	3:
		bTimer1															:= TRUE;
		bPass1															:= steam_bypass_valve_clear;
		bPass2															:= steam_iso_valve_clear;
		bPass3															:= product_iso_valve_clear;
		bPass4															:= r1.fan_vfd_output = 0;
		bPass5															:= P_U01.vacuum_pres_control_valve_closed;
		bPass6															:= P_U01.steam_flow_control_valve_closed;
		bPass7															:= P_U01.product_line_ambient_valve_clear;
		bPass8															:= P_U01.vacuum_pump_bypass_valve_clear;
		bPass9															:= P_U01.vacuum_pump_inlet_valve_clear;
		IF bPass1 AND bPass2 AND bPass3 AND bPass4 AND bPass5 AND bPass6 AND bPass7 AND bPass8 AND bPass9 THEN
			bTimer1														:= FALSE;
			rTime1														:= _SECONDS * 60;
			i6Step														:= i6Step + 1;
		ELSIF tonTimer1.Q THEN
			bTimer1														:= FALSE;
			sReactorError												:= SEL(bPass1,'Steam Bypass Valve Error RS XV08', '');
			sReactorError												:= SEL(bPass2, gsSteamIsoValveError, sReactorError);
			sReactorError												:= SEL(bPass3, gsProductIsoValveError, sReactorError);
			sReactorError												:= SEL(bPass4, 'Fan VFD SP Error', sReactorError);
			sUtilityError												:= SEL(bPass5, gsVacuumPressureControlValveError, '');
			sUtilityError												:= SEL(bPass6, gsSteamFlowConrolValveError, sUtilityError);
			sUtilityError												:= SEL(bPass7, gsProductLineAmbientValveError, sUtilityError);
			sUtilityError												:= SEL(bPass8, gsVacuumPumpBypassValveError, sUtilityError);
			sUtilityError												:= SEL(bPass9, gsVacuumPumpInletValveError, sUtilityError);
		END_IF
		
	4:
		bTimer1															:= TRUE;
		bPass1															:= r1.reactor_pres > P_M01.SP_evacuation_ideal_pressure;
		bPass2															:= NOT reactor_drain_vessel_lsh;
		bPass3															:= NOT P_U01.product_condensate_drum_lsh;
//		bPass4															:= P_U01.vacuum_separator_level > P_U01.SP_vacuum_separator_level_low;
		IF bPass1 AND bPass2 AND bPass3  THEN
			bTimer1														:= FALSE;
			cycle_stage													:= 'evacuation.starting';
			P_U01.drainage_on											:= FALSE;											
			i6Step														:= i6Step + 1;
		ELSIF tonTimer1.Q THEN
			bTimer1														:= FALSE;
			sReactorError												:= SEL(bPass1, gsReactorPressureTooLowError, '');
			sReactorError												:= SEL(bPass2, gsReactorDrainError, sReactorError);
			sUtilityError												:= SEL(bPass3, gsProductCondensateDrumLshError, '');
		END_IF
	
	5:
		
			rTime1														:= _CLAMP_ACTUATION_TIMEOUT;
			P_U01.vacuum_liquid_pump									:= TRUE;											
			P_U01.vacuum_liquid_loop_fan								:= TRUE;
			retract_clamps												:= TRUE;											
			i6Step														:= i6Step + 1;
		
	6:
		bTimer1															:= TRUE;
		IF inlet_clamps_retracted AND outlet_clamps_retracted THEN
			bTimer1														:= FALSE;
			close_doors													:= TRUE;											
			rTime1														:= _DOOR_ACTUATION_TIMEOUT;
			i6Step														:= i6Step + 1;
		ELSIF tonTimer1.Q THEN
			bTimer1														:= FALSE;
			sReactorError												:= SEL(inlet_clamps_retracted, gsInletDoorClampsRetractedError, '');
			sReactorError												:= SEL(outlet_clamps_retracted, gsOutletDoorClampsRetractedError, sReactorError);
		END_IF

	7:
		bTimer1															:= TRUE;
		IF inlet_doors_closed AND outlet_doors_closed THEN
			bTimer1														:= FALSE;
			extend_clamps												:= TRUE;											
			rTime1														:= 30 * _SECONDS;
			i6Step														:= i6Step + 1;
		ELSIF tonTimer1.Q THEN
			sReactorError												:= gsDoorsNotClosedError;
			bTimer1														:= FALSE;
		END_IF

	8:
		cycle_stage														:= 'evacuation.vacuum_init';
		bTimer1															:= TRUE;
		bPass1															:= P_U01.vacuum_pump_water_flow > P_U01.SP_minimum_vacuum_cooling_loop_flow;
		bPass2															:= P_U01.vacuum_pump_water_temp_1 < P_U01.SP_max_vacuum_cooling_loop_temp;
		IF bPass1 AND bPass2 THEN																							
			bTimer1														:= FALSE;
			cycle_stage													:= 'evacuation.evacuation';
			P_U01.dead_air_inlet_valve									:= TRUE;
			P_U01.vacuum_pump											:= TRUE;
			rTime1														:= 20 * _SECONDS;
			i6Step														:= i6Step + 1;
		ELSIF tonTimer1.Q THEN
			bTimer1														:= FALSE;
			sUtilityError												:= SEL(bPass1, gsVacuumCoolingLoopFlowError, '');
			sUtilityError												:= SEL(bPass2, gsVacuumCoolingLoopTempError, sUtilityError);
		END_IF
			
	9:
		bTimer1															:= TRUE;
		bPass1															:= P_U01.product_vacuum_pres <= P_U01.SP_minimum_dead_air_line_pressure;
		IF P_U01.dead_air_inlet_valve_clear AND bPass1 THEN
			bTimer1														:= FALSE;						
			dead_air_valve												:= TRUE;
			rTime1														:= _VALVE_TIME;
			i6Step														:= i6Step + 1;
		ELSIF tonTimer1.Q THEN
			bTimer1														:= FALSE;
			sUtilityError												:= SEL(P_U01.dead_air_inlet_valve_clear,gsDeadAirInletValveError,'');
			sUtilityError												:= SEL(bPass1,gsDeadAirLinePressureError,sUtilityError);
		END_IF
	
	10:
		bTimer1															:= TRUE;	
		IF dead_air_valve_clear	THEN
			bTimer1														:= FALSE;
			rTime1														:= P_M01.SP_evacuation_duration * _MINUTES;
			i6Step														:= i6Step + 1;
		ELSIF tonTimer1.Q THEN
			sReactorError												:= gsDeadAirValveError;
			bTimer1														:= FALSE;
		END_IF
	
	11:
		bTimer1															:= TRUE;
		IF r1.reactor_pres <= P_M01.SP_evacuation_ideal_pressure  THEN														
			bTimer1														:= FALSE;
//			rReactorLeakTestStartingPressure							:= r1.reactor_pres;
			dead_air_valve												:= FALSE;
			P_U01.dead_air_inlet_valve									:= FALSE;
			P_U01.vacuum_pump											:= FALSE;
			P_U01.vacuum_liquid_pump									:= FALSE;
			P_U01.vacuum_liquid_loop_fan								:= FALSE;
			rTime1														:= _VALVE_TIME;
			i6Step														:= i6Step + 1;
		ELSIF tonTimer1.Q THEN
			bTimer1														:= FALSE;
			sReactorError												:= gsReactorPressureTooHighError;
		END_IF
		
	12:
		bTimer1															:= TRUE;
		IF dead_air_valve_clear AND P_U01.dead_air_inlet_valve_clear  AND inlet_clamps_extended AND outlet_clamps_extended THEN																						// 10
			bTimer1														:= FALSE;
			rTime1														:= P_M01.SP_vacuum_leak_test_duration * _MINUTES;
			i6Step														:= i6Step + 1;
		ELSIF tonTimer1.Q THEN
			bTimer1														:= FALSE;
			sReactorError												:= SEL(dead_air_valve_clear,gsDeadAirValveError,'');
			sUtilityError												:= gsDeadAirInletValveError;
			sReactorError												:= SEL(inlet_clamps_extended, gsInletDoorClampsExtendedError, '');
			sReactorError												:= SEL(outlet_clamps_extended, gsOutletDoorClampsExtendedError, sReactorError);
		END_IF
		
	13: //mm
		bTimer1															:= TRUE;
		IF tonTimer1.Q THEN
//			reactor_test_leakage_pressure									:= r1.reactor_pres - rReactorLeakTestStartingPressure;
			IF r1.reactor_pres  <= P_M01.SP_evacuation_ideal_pressure * 1.1 THEN									// 11
				bTimer1													:= FALSE;
				rTime1													:= _STOPPING_TIME;
				i6Step													:= 98;
			ELSE
				bTimer1													:= FALSE;
				sReactorError											:= gsUnacceptableReactorLeakRate;
			END_IF
		END_IF
		
	

	80:																														// Stop process individually 
		cycle_stage														:= 'evacuation.stopping';
		dead_air_valve													:= FALSE;											
		P_U01.dead_air_inlet_valve										:= FALSE;
		P_U01.vacuum_pump												:= FALSE;
		P_U01.vacuum_liquid_pump										:= FALSE;
		P_U01.vacuum_liquid_loop_fan									:= FALSE;
		A_Reset();
		rTime1															:= _STOPPING_TIME;
		i6Step															:= 98;
		
	90:																														// Automatic process stopping
		cycle_stage														:= 'evacuation.stopping';
		A_Reset();
		rTime1															:= _STOPPING_TIME;
		i6Step															:= 98;
		
	98:
		cycle_stage														:= 'evacuation.stopping';
		bTimer1															:= TRUE;
		IF tonTimer1.Q THEN
			bTimer1														:= FALSE;
			i6Step														:= 99;
		END_IF
		
	99:
		bEvacuationDone													:= TRUE;											// 13
		Current_Step													:= 0;
		i6Step															:= 0;
	
END_CASE

IF i6Step > 0 AND i6Step < 80 THEN
	iStep																:= i6Step;
	Current_Step														:= iStep;
	sReactorError														:= SEL(r1.reactor_pres_error, sReactorError, gsReactorPresSensorError);
	sUtilityError														:= SEL(P_U01.vacuum_separator_level_error, sUtilityError, gsVacuumSeparatorLevelSensorError);
	sUtilityError														:= SEL(P_U01.vacuum_pump_water_flow_error, sUtilityError, gsVacuumPumpWaterFlowSensorError);
	sUtilityError														:= SEL(P_U01.vacuum_pump_water_temp_1_error, sUtilityError, gsVacuumPumpWaterTemp1SensorError);
	A_Check_Process();
	i6Step																:= iStep;
END_IF
END_ACTION

ACTION A6_Evacuation_1:

CASE i6Step OF	

	0:	;
		
	1:
		cycle_stage														:= 'evacuation.initialize';
		rTime1															:= _VALVE_TIME;
		i6Step															:= i6Step + 1;
		
	2:
		cycle_stage														:= 'evacuation.started';
		bTimer1															:= TRUE;
		IF tonTimer1.Q THEN
			bTimer1														:= FALSE;
			i6Step														:= 98;
		END_IF
		
	80:																														// Stop process individually 
		cycle_stage														:= 'evacuation.stopping';
		rTime1															:= _STOPPING_TIME;
		i6Step															:= 98;
		
	90:																														// Automatic process stopping
		cycle_stage														:= 'evacuation.stopping';
		rTime1															:= _STOPPING_TIME;
		i6Step															:= 98;
		
	98:
		cycle_stage														:= 'evacuation.stopping';
		bTimer1															:= TRUE;
		IF tonTimer1.Q THEN
			bTimer1														:= FALSE;
			i6Step														:= 99;
		END_IF
	99:
		cycle_stage														:= 'evacuation.completed';
		bEvacuationDone													:= TRUE;											// 5
		Current_Step													:= 0;
		i6Step															:= 0;
	
END_CASE

IF i6Step > 0 AND i6Step < 80 THEN
	iStep																:= i6Step;
	Current_Step														:= iStep;
	A_Check_Process();
	i6Step																:= iStep;
END_IF
END_ACTION

ACTION A6_Evacuation_OLD:
// Theseus - FB_Reactor_Set.A6_Evacuation
// Rev 1.0 - October 9, 2024

CASE i6Step OF
	
	0:	;
	
	1:
		cycle_stage														:= 'evacuation.initialize';
		giEvacuationCounter												:= giEvacuationCounter - 1;
		sMessage														:= gsSystemCannotRun;
		gbGasketsActivated												:= FALSE;
		IF P_U01.utility_error <> '' THEN
			sUtilityError												:= P_U01.utility_error;
		ELSIF product_line_pres_error THEN
			sReactorError												:= gsProductLinePressureSensorError;
		ELSIF r1.reactor_pres_error THEN
			sReactorError												:= gsReactorPresSensorError;
		ELSIF inlet_clamps_extended AND outlet_clamps_extended THEN
			i6Step														:= i6Step + 3;
			rTime1														:= 1 * _SECONDS;
		ELSE
			A_Reset();																										// 1
			retract_clamps												:= TRUE;											// 2
			rTime1														:= _CLAMP_ACTUATION_TIMEOUT; 		// Use Valve time if longer
			i6Step														:= i6Step + 1;
		END_IF
		
	2:
		bTimer1															:= TRUE;
		cycle_stage														:= 'evacuation.close_valve_doors';
		IF rs_valves_clear AND inlet_clamps_extended AND outlet_clamps_extended THEN
			bTimer1														:= FALSE;
			close_doors													:= TRUE;
			rTime1														:= _DOOR_ACTUATION_TIMEOUT;
			i6Step														:= i6Step + 1;
		ELSIF tonTimer1.Q THEN
			IF inlet_clamps_extended AND outlet_clamps_extended THEN
				sReactorError											:= SEL(dead_air_valve_clear, gsDeadAirValveError, '');
				sReactorError											:= SEL(product_iso_valve_clear, gsProductIsoValveError, sReactorError);
				sReactorError											:= SEL(condensate_valve_clear, gsCondensateValveError, sReactorError);
				sReactorError											:= SEL(steam_iso_valve_clear, gsSteamIsoValveError, sReactorError);
				sReactorError											:= SEL(steam_bypass_valve_clear, gsSteamBypassValveError, sReactorError);
			ELSE
				sReactorError											:= SEL(NOT inlet_clamps_extended, '', gsInletDoorClampsExtendedError);
				sReactorError											:= SEL(outlet_clamps_extended, sReactorError, gsOutletDoorClampsExtendedError);
			END_IF
		END_IF

	3:
		bTimer1															:= TRUE;
		IF (inlet_doors_closed AND outlet_doors_closed) OR r1.reactor_pres < 0.9 THEN				// smrg debug - allow test to continue if picking up where previous vacuum test left off (doors may not show up as closed under vacuum)
			bTimer1														:= FALSE;
			extend_clamps												:= TRUE;
			rTime1														:= _CLAMP_ACTUATION_TIMEOUT;
			i6Step														:= i6Step + 1;
		ELSIF tonTimer1.Q THEN
			sReactorError												:= gsDoorsNotClosedError;
		END_IF

	4:
		bTimer1															:= TRUE;
		IF tonTimer1.Q THEN
			bTimer1														:= FALSE;
			P_U01.dead_air_inlet_valve									:= TRUE;											// 5
			P_U01.product_line_ambient_valve							:= INT_TO_BOOL(eAmbient);	
			P_U01.vacuum_liquid_loop_fan								:= TRUE;
			P_U01.vacuum_liquid_pump									:= TRUE;
			repres_valves												:= FALSE;
			steam_iso_valve												:= FALSE;
			rTime1														:= 5 * _SECONDS;									// give water time to start flowing before attempting to turn on vacuum pump
			i6Step														:= i6Step + 1;
		END_IF
		
	5:
		bTimer1															:= TRUE;
		IF tonTimer1.Q THEN
			bTimer1														:= FALSE;
			rTime1														:= _VALVE_TIME;
			i6Step														:= i6Step + 1;
		END_IF
		
	6:		
		cycle_stage														:= 'evacuation.vacuum_init';
		bTimer1															:= TRUE;
		//IF P_U01.dead_air_inlet_valve_clear AND P_U01.product_line_ambient_valve_clear THEN
		IF P_U01.dead_air_inlet_valve_clear THEN								// smrg debug
			bTimer1														:= FALSE;
			P_U01.vacuum_pump											:= TRUE;											// 6
			cycle_stage													:= 'evacuation.evacuation';
			rTime1														:= 60 * _SECONDS;
			i6Step														:= i6Step + 1;
		ELSIF tonTimer1.Q THEN
			sReactorError												:= SEL(dead_air_valve_clear, gsDeadAirValveError, '');
			sReactorError												:= SEL(P_U01.product_line_ambient_valve_clear, gsProductLineAmbientValveError, sReactorError);
		END_IF
		
	7:
		bTimer1															:= TRUE;
		IF P_U01.product_vacuum_pres <= P_M01.SP_evacuation_ideal_pressure THEN													// 7
			bTimer1														:= FALSE;
			dead_air_valve												:= TRUE;											// 8		
			rTime1														:= _VALVE_TIME;
			i6Step														:= i6Step + 1;
		ELSIF tonTimer1.Q THEN
			sReactorError												:= gsDeadAirValveError;
		END_IF
		
	8:
		bTimer1															:= TRUE;
		IF dead_air_valve_clear THEN													
			rTime1														:= P_M01.SP_evacuation_duration * _MINUTES;
			bTimer1														:= FALSE;										
			i6Step														:= i6Step + 1;
		ELSIF tonTimer1.Q THEN
			sReactorError												:= gsVacuumLinePressureHighError;
		END_IF
	
	9:
		bTimer1															:= TRUE;
		IF r1.reactor_pres <= P_M01.SP_evacuation_ideal_pressure THEN														// 9
			bTimer1														:= FALSE;
			i6Step														:= i6Step + 1;
		ELSIF tonTimer1.Q THEN
			sReactorError												:= gsReactorPressureTooHighError;
		END_IF

	10:
		IF inlet_clamps_extended AND outlet_clamps_extended THEN																						
			gbGasketsActivated											:= TRUE;											// 10
			dead_air_valve												:= FALSE;											// 11
			P_U01.vacuum_liquid_loop_fan								:= FALSE;
			P_U01.vacuum_liquid_pump									:= FALSE;
			P_U01.vacuum_pump											:= FALSE;
			rTime1														:= _VALVE_TIME;
			i6Step														:= i6Step + 1;
		ELSE
			sReactorError												:= SEL(NOT inlet_clamps_extended, '', gsInletDoorClampsExtendedError);
			sReactorError												:= SEL(NOT outlet_clamps_extended, sReactorError, gsOutletDoorClampsExtendedError);
		END_IF		
		
	11:
		bTimer1															:= TRUE;
		IF dead_air_valve_clear THEN
			bTimer1														:= FALSE;
			IF gbFirstEvacuation THEN																						// 12
				gbFirstEvacuation										:= FALSE;
				cycle_stage												:= 'evacuation.settle_time';
				rTime1													:= P_M01.SP_vacuum_settle_time * _MINUTES;			// 13
				i6Step													:= i6Step + 1;
			ELSE																											// if not first evacuation, skip leak check
				i6Step													:= 13;
			END_IF
		ELSIF tonTimer1.Q THEN
			sReactorError												:= gsDeadAirValveError;
		END_IF

	12:
		bTimer1															:= TRUE;
		IF tonTimer1.Q THEN	
			bTimer1														:= FALSE;			
			cycle_stage													:= 'evacuation.leak_check';
			rR1SavedPressure											:= r1.reactor_pres;									// 14
			rTime1														:= P_M01.SP_vacuum_leak_test_duration * _MINUTES;
			i6Step														:= i6Step + 1;
		END_IF
		
	13:
		bTimer1															:= TRUE;
		IF tonTimer1.Q THEN																									// 15
			bTimer1														:= FALSE;
			rR1Leakage													:= (r1.reactor_pres - rR1SavedPressure) / P_M01.SP_vacuum_leak_test_duration;
			IF rR1Leakage < P_M01.SP_unacceptable_vacuum_pressure_change THEN												// 16
				bVacuumHolding											:= TRUE;
				i6Step													:= i6Step + 1;
			ELSE
				bVacuumHolding											:= FALSE;
				sReactorError											:= gsVacuumPressureUnacceptableError;
			END_IF
		END_IF

	14:
		IF (giEvacuationCounter = 0) THEN																					// 17
			retract_clamps												:= TRUE;											// 18
			rTime1														:= _CLAMP_ACTUATION_TIMEOUT;
			i6Step														:= i6Step + 1;
		ELSE
			i6Step														:= 99;
		END_IF
 
	15:
		bTimer1															:= TRUE;
		IF inlet_clamps_retracted AND outlet_clamps_retracted THEN
			i6Step														:= 99;
		ELSIF tonTimer1.Q THEN
			sReactorError												:= gsDoorClampsExtendedError;
			sMessage													:= gsSystemWillStop;
		END_IF
		
	80:																														// Stop process
		cycle_stage														:= 'evacuation.stopping';
		A_Reset();
		rTime1															:= _STOPPING_TIME;
		i6Step															:= 98;
		
	90:																														// Automatic process stopping
		cycle_stage														:= 'evacuation.stopping';
		A_Reset();
		rTime1															:= _STOPPING_TIME;
		i6Step															:= 98;
		
	98:
		bTimer1															:= TRUE;
		IF tonTimer1.Q THEN
			bTimer1														:= FALSE;
			i6Step														:= 99;
		END_IF
		
	99:
		bEvacuationDone													:= TRUE;											// 19
		Current_Step													:= 0;
		i6Step															:= 0;
	
END_CASE

IF i6Step > 0 AND i6Step < 80 THEN
	iStep																:= i6Step;
	Current_Step														:= iStep;
	A_Check_Process();
	i6Step																:= iStep;
END_IF
END_ACTION

ACTION A7_Desorption:
// Theseus - FB_Reactor_Set.A7_Desorption_1
// Rev 1.0 - June 24, 2024

CASE i7Step OF
	
	0:	;
		
	1:
		
		cycle_stage														:= 'desorption.initialize';
		sMessage														:= gsSystemCannotRun;
		
		IF P_U01.utility_error <> '' THEN
			sUtilityError												:= P_U01.utility_error;
		ELSIF r1.reactor_pres_error THEN
			sReactorError												:= gsReactorPresSensorError;
		ELSE			
			A_Reset();
			P_U01.boiler_package 										:= FALSE;
//			P_U01.vacuum_pres_control_valve								:= _CLOSED;											//add it as input to P_U01			
			rTime1															:= _VALVE_TIME;
			i7Step															:= i7Step + 1;										
		END_IF		
		
		
	2:
		rTime1															:= _VALVE_TIME;
		bTimer1															:= TRUE;
		IF rs_valves_clear AND P_U01.vacuum_pres_control_valve_closed  THEN
			bTimer1														:= FALSE; 
			i7Step														:= i7Step + 1;
		ELSIF tonTimer1.Q THEN
			sReactorError												:= gsProcessCannotContinue;
		END_IF	
	
	3: //excel sheet step2 - open repres valve
		cycle_stage														:= 'desorption.running';
		r1.repres_valve													:= TRUE;
		rTime1															:= _VALVE_TIME;
		bTimer1															:= TRUE;
		IF R1.repres_valve_clear THEN
			bTimer1														:= FALSE;
			i7Step														:= i7Step + 1;
		ELSIF tonTimer1.Q THEN
			sReactorError												:= gsRepressurizationValveError;
		END_IF

	4: //excel sheet step 3 - wait for repressurization
		rTime1															:= 5 * _MINUTES;
		bTimer1															:= TRUE;
		IF r1.reactor_pres > 0.98 AND r1.reactor_pres < 1.02 THEN
			bTimer1														:= FALSE;
			i7Step														:= i7Step + 1;
		ELSIF tonTimer1.Q THEN
			sReactorError												:= gsRepressurizationError;
		END_IF
		
	5: //excel sheet step 4 - settle time
		rTime2															:=10 * _SECONDS;
		bTimer2															:= TRUE;
		IF tonTimer2.Q THEN
			bTimer2														:= FALSE;
			i7Step														:= 99;
		END_IF
		
	80:																														// Manual process completing
		cycle_stage														:= 'desorption.stopping';
		rTime1															:= _STOPPING_TIME;
		A_Reset();
		i7Step															:= 98;
		
	90:																														// Automatic process completing 
		cycle_stage														:= 'desorption.stopping';
		rTime1															:= _STOPPING_TIME;
		A_Reset();
		i7Step															:= 98;
		
	98:
		bTimer1															:= TRUE;
		IF tonTimer1.Q THEN
			bTimer1														:= FALSE;
			i7Step														:= 99;
		END_IF
			
		
	99:
		bDesorptionDone													:= TRUE;											// 19
		Current_Step													:= 0;
		i7Step															:= 0;
	
END_CASE

IF i7Step > 0 AND i7Step < 80 THEN
	iStep																:= i7Step;
	Current_Step														:= iStep;
	A_Check_Process();
	i7Step																:= iStep;
END_IF
END_ACTION

ACTION A7_Desorption_1:
// Theseus - FB_Reactor_Set.A7_Desorption_1
// Rev 1.0 - June 24, 2024

CASE i7Step OF
	
	0:	;
		
	1:
		rTime1															:= _VALVE_TIME;
		i7Step															:= i7Step + 1;
		
	2:
		bTimer1															:= TRUE;
		IF tonTimer1.Q THEN
			bTimer1														:= FALSE;
			i7Step														:= 99;
		END_IF

	99:
		bDesorptionDone													:= TRUE;											// 19
		Current_Step													:= 0;
		i7Step															:= 0;
	
END_CASE

IF i7Step > 0 AND i7Step < 80 THEN
	iStep																:= i7Step;
	Current_Step														:= iStep;
	A_Check_Process();
	i7Step																:= iStep;
END_IF
END_ACTION

ACTION A7_Desorption_OLD:
// Theseus - FB_Reactor_Set.A7_Desorption
// Rev 1.0 - June 17, 2024

CASE i7Step OF
	
	0:	;
		
	1:
		i7Step															:= 0;
	
END_CASE

IF i7Step > 0 AND i7Step < 80 THEN
	iStep																:= i7Step;
	Current_Step														:= iStep;
	A_Check_Process();
	i7Step																:= iStep;
END_IF
END_ACTION

ACTION A8_Bypass:
// Theseus - FB_Reactor_Set.A8_Bypass
// Rev 1.0 - December 3, 2024

CASE i8Step OF
	
	0:	;
	
	1:
		cycle_stage														:= 'bypass.initialize';
		sMessage														:= gsSystemCannotRun;
		i8Step															:= i8Step + 1;										// Run first step to check for sensor errors
		
	2:
		A_Reset();																											// 1
		P_U01.vacuum_pres_control_valve_mode							:= eManual;
		P_U01.vacuum_pres_control_valve									:= _CLOSED;
		P_U01.steam_flow_control_valve_mode								:= eManual;
		P_U01.steam_flow_control_valve									:= _CLOSED;
		P_U01.product_line_ambient_valve								:= FALSE;
		P_U01.vacuum_pump_inlet_valve									:= FALSE;
		P_U01.vacuum_pump_bypass_valve									:= TRUE;
		P_U01.drainage_on												:= TRUE;
		rTime1															:= _VALVE_TIME;
		i8Step															:= i8Step + 1;
		
	3:
		bTimer1															:= TRUE;
		bPass1															:= P_U01.vacuum_pres_control_valve_closed;
		bPass2															:= P_U01.steam_flow_control_valve_closed;
		bPass3															:= P_U01.product_line_ambient_valve_clear;
		bPass4															:= P_U01.vacuum_pump_inlet_valve_clear;
		bPass5															:= P_U01.vacuum_pump_bypass_valve_clear;
		IF rs_valves_clear AND bPass1 AND bPass2 AND bPass3 AND bPass4 AND bPass5 THEN
			bTimer1														:= FALSE;
			IF P_U01.boiler_ready THEN																						// 2
				P_U01.condenser_fan										:= TRUE;
				P_U01.condenser_pump									:= TRUE;
				P_U01.steam_flow_control_valve_mode						:= eManual;											// 3
				P_U01.steam_flow_control_valve							:= _OPEN;
				steam_bypass_valve										:= TRUE;
				rTime1													:= _VALVE_TIME;
				i8Step													:= i8Step + 1;
			ELSE
				sUtilityError											:= gsBoilerError;
			END_IF
		ELSIF tonTimer1.Q THEN
			bTimer1														:= FALSE;
			sReactorError												:= SEL(dead_air_valve_clear, gsDeadAirValveError, '');
			sReactorError												:= SEL(product_iso_valve_clear, gsProductIsoValveError, sReactorError);
			sReactorError												:= SEL(condensate_valve_clear, gsCondensateValveError, sReactorError);
			sReactorError												:= SEL(steam_iso_valve_clear, gsSteamIsoValveError, sReactorError);
			sReactorError												:= SEL(steam_bypass_valve_clear, gsSteamBypassValveError, sReactorError);
			sUtilityError												:= SEL(bPass1, gsVacuumPressureControlValveError, '');
			sUtilityError												:= SEL(bPass2, gsSteamFlowConrolValveError, sUtilityError);
			sUtilityError												:= SEL(bPass3, gsProductLineAmbientValveError, sUtilityError);
			sUtilityError												:= SEL(bPass4, gsVacuumPumpInletValveError, sUtilityError);
			sUtilityError												:= SEL(bPass5, gsVacuumPumpBypassValveError, sUtilityError);
		END_IF
		
	4:
		bTimer1															:= TRUE;
		bPass1															:= P_U01.steam_flow_control_valve_open;
		bPass2															:= steam_bypass_valve_clear;
		IF bPass1 AND bPass2 THEN
			bTimer1														:= FALSE;
			cycle_stage													:= 'bypass.running';
			rTime1														:= P_U01.SP_minimum_steam_bypass_duration * _MINUTES;
			i8Step														:= i8Step + 1;
		ELSIF tonTimer1.Q THEN
			bTimer1														:= FALSE;
			sUtilityError												:= SEL(bPass1, gsSteamFlowConrolValveError, '');
			sReactorError												:= SEL(bPass2, gsSteamBypassValveError, '');
		END_IF
		
	5:	bTimer1															:= TRUE;
		IF tonTimer1.Q THEN
			bTimer1														:= FALSE;
			bPass1														:= P_U01.steam_flow > P_U01.SP_minimum_steam_bypass_flow_rate;
			bPass2														:= product_line_temp > 90;
			IF bPass1 AND bPass2 THEN
				steam_bypass_valve										:= FALSE;											// 4
				P_U01.steam_flow_control_valve_mode						:= eManual;											///@@@ Not specified in narrative
				P_U01.steam_flow_control_valve							:= _CLOSED;
				rTime1													:= _VALVE_TIME;										// 5
				i8Step													:= i8Step + 1;
			ELSE
				sUtilityError											:= SEL(bPass1, gsSteamFlowTooLowError, '');
				sReactorError											:= SEL(bPass2, gsProductLineTempTooLowError, '');
			END_IF
		END_IF

	6:
		bTimer1															:= TRUE;
		bPass1															:= P_U01.steam_flow_control_valve_closed;
		bPass2															:= steam_bypass_valve_clear;
		IF bPass1 AND bPass2 THEN
			bTimer1														:= FALSE;
			P_U01.vacuum_pump_bypass_valve								:= FALSE;											// 6
			P_U01.product_line_ambient_valve							:= TRUE;
			rTime1														:= _VALVE_TIME;
			i8Step														:= i8Step + 1;
		ELSIF tonTimer1.Q THEN
			bTimer1														:= FALSE;
			sUtilityError												:= SEL(bPass1, gsSteamFlowConrolValveError, '');
			sReactorError												:= SEL(bPass2, gsSteamBypassValveError, '');
		END_IF

	7:
		bTimer1															:= TRUE;
		bPass1															:= P_U01.product_line_ambient_valve_clear;
		bPass2															:= P_U01.vacuum_pump_bypass_valve_clear;
		IF bPass1 AND bPass2 THEN
			bTimer1														:= FALSE;
			i8Step														:= 99;
		ELSIF tonTimer1.Q THEN
			bTimer1														:= FALSE;
			sUtilityError												:= SEL(bPass1, gsProductLineAmbientValveError, '');
			sUtilityError												:= SEL(bPass2, gsVacuumPumpBypassValveError, sUtilityError);
		END_IF
		
	80:																														// Stop process
		cycle_stage														:= 'bypass.stopping';
		A_Reset();
		P_U01.drainage_on												:= FALSE;
		P_U01.vacuum_pump_bypass_valve									:= FALSE;
		P_U01.condenser_fan												:= FALSE;
		P_U01.condenser_pump											:= FALSE;
		P_U01.steam_flow_control_valve_mode								:= eManual;
		P_U01.steam_flow_control_valve									:= _CLOSED;
		P_U01.product_line_ambient_valve								:= FALSE;											///@@@ Correct position???
		rTime1															:= _STOPPING_TIME;
		i8Step															:= 98;
		
	90:																														// Automatic process stopping
		cycle_stage														:= 'bypass.stopping';
		A_Reset();
		rTime1															:= _STOPPING_TIME;
		i8Step															:= 98;
		
	98:
		bTimer1															:= TRUE;
		IF tonTimer1.Q THEN
			bTimer1														:= FALSE;
			i8Step														:= 99;
		END_IF
		
	99:
		bBypassDone														:= TRUE;											// 13
		Current_Step													:= 0;
		i8Step															:= 0;
	
END_CASE

IF i8Step > 0 AND i8Step < 80 THEN
	iStep																:= i8Step;
	Current_Step														:= iStep;
	sReactorError														:= SEL(product_line_temp_error, sReactorError, gsProductLineTempSensorError);
	sUtilityError														:= SEL(P_U01.steam_flow_error, sUtilityError, gsSteamFlowSensorError);
	A_Check_Process();
	i8Step																:= iStep;
END_IF
END_ACTION

ACTION A8_Bypass_1:
CASE i8Step OF	

	0:	;
		
	1:
		rTime1															:= _VALVE_TIME;
		i8Step															:= i8Step + 1;
		
	2:
		bTimer1															:= TRUE;
		IF tonTimer1.Q THEN
			bTimer1														:= FALSE;
			i8Step														:= 99;
		END_IF
	
	99:
		bBypassDone														:= TRUE;											// 5
		Current_Step													:= 0;
		i8Step															:= 0;
	
END_CASE

IF i8Step > 0 AND i8Step < 80 THEN
	iStep																:= i8Step;
	Current_Step														:= iStep;
	A_Check_Process();
	i8Step																:= iStep;
END_IF
END_ACTION

END_FUNCTION_BLOCK

// ---- POUs/Function_Blocks/FB_ChangeOfValue.TcPOU
FUNCTION_BLOCK FB_ChangeOfValue
VAR_INPUT
	i_execute		: BOOL;
	i_value			: REAL;
	i_time			: REAL;
	i_threshold			: REAL;
END_VAR
VAR_OUTPUT
	o_delta				: REAL;
	o_below_threshold	: BOOL;
	o_timeout			: BOOL;
END_VAR
VAR
	tmrSampleTime	: TON;
	state			: (idle, first_cycle,second_cycle);
	rtrig_execute	: R_TRIG;
	value_first_cycle	: REAL;
	value_second_cycle	: REAL;
	old_value : REAL;
	new_value : REAL;
	delta_value : REAL;
	tmrTimeout : TON;
END_VAR

rtrig_execute(CLK := i_execute);
(*
IF NOT i_execute THEN
	state := idle;
END_IF

CASE state OF
	idle : 	
		tmrSampleTime.IN := FALSE;
		IF rtrig_execute.Q THEN 
			o_oor := FALSE;
			o_delta := 0;
//			state := first_cycle;
			
		END_IF
	first_cycle: 
		value_first_cycle := i_value;
		tmrSampleTime.IN := TRUE;
		state := second_cycle;
	second_cycle:
		IF tmrSampleTime.Q THEN
			value_second_cycle := i_value;
			o_delta := ABS(value_second_cycle - value_first_cycle);
			tmrSampleTime.IN := FALSE;
			IF o_delta < i_range THEN
				o_oor := TRUE;
			ELSE
				o_oor := FALSE;
			END_IF
			state := first_cycle;
		END_IF
		
		
END_CASE
*)

IF rtrig_execute.Q THEN
	old_value := i_value;
	o_below_threshold := FALSE;
	tmrTimeout.IN := TRUE;

END_IF
IF i_execute THEN
	tmrSampleTime.IN := TRUE;
	IF tmrSampleTime.Q THEN
		tmrSampleTime.IN := FALSE;
		new_value := i_value;
		delta_value := ABS(new_value - old_value);
		old_value := new_value;
		o_below_threshold := delta_value < i_threshold;
	END_IF
ELSE
	tmrSampleTime.IN := FALSE;
	tmrTimeout.IN 	:= FALSE;
END_IF

IF tmrTimeout.Q THEN
	o_timeout := TRUE;
ELSE
	o_timeout := FALSE;	
END_IF

tmrSampleTime(PT:= TO_TIME(i_time)*1000);
tmrTimeout(PT := T#600S);

END_FUNCTION_BLOCK

// ---- POUs/P_Alarms.TcPOU
PROGRAM P_Alarms
VAR
	i																	: INT;
	sitaBits : DWORD;
	sitaAlarm : STRING;
	sitaMsg : STRING;
	sitaTmr : STRING;
	sitaRTrig : R_TRIG;
	alarm_number : INT;
END_VAR

// Theseus - P_Alarms
// Rev 1.0 - September 30, 2024

FOR i := 1 TO alarm_number DO 
	IF gsAlarms[i] <> '' THEN 
		P_M01.ts_Alarm			:= gsAlarms[i];
		P_M01.ts_User_Message		:= gsMessages[i];
		P_M01.tb_Alarm_Active		:= TRUE;
		EXIT ;
	END_IF
END_FOR


IF P_M01.tb_Acknowledge_Alarm THEN
	FOR i := 1 TO alarm_number DO 
		IF gsAlarms[i] <> '' THEN                     	    	
			gsAlarms[i] 													:= '';
			gsMessages[i]													:= '';
			EXIT ;
		END_IF
	END_FOR
	P_M01.tb_Acknowledge_Alarm := FALSE;                                	    		
END_IF                                      	    	

IF P_M01.tb_Clear_Alarm_All THEN
	FOR i := 1 TO alarm_number DO                      	    	
		gsAlarms[i] 													:= '';
		gsMessages[i]													:= '';	
		P_M01.tb_Clear_Alarm_All											:= FALSE;		
	END_FOR                                 	    	
END_IF

giAlarmCount := M_GetAlarmsCount(); 

IF giAlarmCount = 0 THEN
	P_M01.ts_Alarm			:= '';
	P_M01.ts_User_Message		:= '';
	P_M01.tb_Alarm_Active		:= FALSE;
	alarm_number			:= 0;
END_IF
                                            	    	
FOR i := 1 TO _ALARM_COUNT DO 
	P_M01.processAlarms[i] := gsAlarms[i];
	P_M01.processAlarmsMessage[i] := gsMessages[i];
END_FOR

sitaRTrig(CLK := sitaBits.0);
IF sitaRTrig.Q THEN 
	M_Add_Alarm('UnitTest-',sitaAlarm,sitaMsg);
	sitaBits.0 := FALSE;
END_IF

METHOD M_Add_Alarm 			: BOOL
VAR_INPUT
	Unit																: STRING;
	Alarm																: STRING;
	Message																: STRING;
END_VAR
VAR
END_VAR
// Theseus - P_Alarms.M_Add_Alarm
// Rev 1.0 - January 31, 2024


IF alarm_number < _ALARM_COUNT THEN
	alarm_number													:= alarm_number + 1;
	gsMessages[alarm_number]										:= Message;
	gsAlarms[alarm_number]											:= CONCAT(Unit, Alarm);
END_IF
M_Add_Alarm															:= TRUE;
END_METHOD

METHOD M_Check_Error : BOOL
VAR_INPUT
	Error_In															: BOOL;
	Latch																: BOOL;
	Unit																: STRING;
	Alarm																: STRING;
	Message																: STRING;
END_VAR
VAR
	Error_Out															: BOOL;
END_VAR
// Theseus - P_Alarms.M_Check_Error
// Rev 1.0 - September 30, 2024

IF P_M01.tb_Auto_Mode_On THEN

	Error_Out																:= Latch;
	IF Error_In THEN
		IF NOT Error_Out THEN
			Error_Out														:= TRUE;
			P_Alarms.M_Add_Alarm(Unit, Alarm, Message);
		END_IF
	ELSE
		Error_Out															:= FALSE;
	END_IF
	M_Check_Error															:= Error_Out;

END_IF
END_METHOD

METHOD M_GetAlarmsCount : INT
VAR
	alarmCount : INT := 0 ;
END_VAR

FOR i := 0 TO alarm_number DO 
	IF gsAlarms[i] <> '' THEN 
		alarmCount := alarmCount + 1;
	END_IF
END_FOR
M_GetAlarmsCount := alarmCount;
END_METHOD

END_PROGRAM

// ---- POUs/P_U01.TcPOU
PROGRAM P_U01
VAR_INPUT
	auto_mode_on														: BOOL;

	shutdown_process													: BOOL;
	{attribute 'OPC.UA.DA' := '1'}  				                
	{attribute 'OPC.UA.DA.Access' := '1'}  				                
	co2_adsorption_interlock											: BOOL;
    /// <summary>PCV01</summary>
	{attribute 'OPC.UA.DA' := '1'}  				                
	vacuum_pres_control_valve											: REAL;
    /// <summary>PCV01</summary>                  	           
	{attribute 'OPC.UA.DA' := '1'}  				                
	vacuum_pres_control_valve_mode										: INT;			
    /// <summary>PCV02</summary>
	{attribute 'OPC.UA.DA' := '1'}  				                
	steam_flow_control_valve											: REAL;
    /// <summary>PCV02</summary>                  	           
	{attribute 'OPC.UA.DA' := '1'}  				                
	steam_flow_control_valve_mode										: INT;			
	{attribute 'OPC.UA.DA' := '1'}  				                
	{attribute 'OPC.UA.DA.Access' := '1'}  				                
	hot_sorbent_for_repressurization_interlock							: BOOL;
	{attribute 'OPC.UA.DA' := '1'}  				                
	{attribute 'OPC.UA.DA.Access' := '1'}  				                
	drainage_on															: BOOL;
	{attribute 'OPC.UA.DA' := '1'}  				                
	{attribute 'OPC.UA.DA.Access' := '1'}  				                
	repressurization_valve_with_steam_interlock							: BOOL;
	{attribute 'OPC.UA.DA' := '1'}  				                
	{attribute 'OPC.UA.DA.Access' := '1'}  				                
	door_open_with_steam_flow_interlock									: BOOL;
	{attribute 'OPC.UA.DA' := '1'}  				                
	{attribute 'OPC.UA.DA.Access' := '1'}  				                
	door_open_with_reactor_vacuum_interlock								: BOOL;
	{attribute 'OPC.UA.DA' := '1'}  				                
	{attribute 'OPC.UA.DA.Access' := '1'}  				                
	hot_reactor_condenser_interlock										: BOOL;
	{attribute 'OPC.UA.DA' := '1'}  				                
	{attribute 'OPC.UA.DA.Access' := '1'}  				                
	no_steam_unevacuated_reactor_interlock								: BOOL;
	{attribute 'OPC.UA.DA' := '1'}  				                
	{attribute 'OPC.UA.DA.Access' := '1'}  				                
	reactor_over_safe_pressure_limit_interlock							: BOOL;
	{attribute 'OPC.UA.DA' := '1'}  				                
	{attribute 'OPC.UA.DA.Access' := '1'}  				                
	reactor_over_safe_temperature_limit_interlock						: BOOL;
	
	/// <summary>XV10</summary>
	{attribute 'OPC.UA.DA' := '1'}  				                
	dead_air_inlet_valve												: BOOL;
	/// <summary>XV11</summary>
	{attribute 'OPC.UA.DA' := '1'}  				                
	product_line_ambient_valve											: BOOL;
    /// <summary>X01</summary>
	{attribute 'OPC.UA.DA' := '1'}  				                
	vacuum_liquid_loop_fan												: BOOL;
    /// <summary>P05</summary>
	{attribute 'OPC.UA.DA' := '1'}  				                
	vacuum_liquid_pump													: BOOL;
    /// <summary>P02</summary>
	{attribute 'OPC.UA.DA' := '1'}  				                
	vacuum_pump															: BOOL;
    /// <summary>XV04</summary>
	{attribute 'OPC.UA.DA' := '1'}  				                
	vacuum_pump_bypass_valve											: BOOL;
    /// <summary>XV03</summary>
	{attribute 'OPC.UA.DA' := '1'}  				                
	vacuum_pump_inlet_valve												: BOOL;
    /// <summary>P01</summary>
	{attribute 'OPC.UA.DA' := '1'}  				                
	steam_water_pump													: BOOL;
    /// <summary>B01</summary>
	{attribute 'OPC.UA.DA' := '1'}  				                
	boiler_package														: BOOL;
    /// <summary>P04</summary>
	{attribute 'OPC.UA.DA' := '1'}  				                
	condenser_pump														: BOOL;
    /// <summary>E01</summary>
	{attribute 'OPC.UA.DA' := '1'}  				                
	condenser_fan														: BOOL;
    /// <summary>P06</summary>
	{attribute 'OPC.UA.DA' := '1'}  				                
	vacuum_separator_drain_pump											: BOOL;
    /// <summary>PCV02</summary>
	steam_flow_control_valve_setpoint									: REAL;
	condenser_knockout_drain_adsorption_on									: BOOL;
	
END_VAR
VAR_OUTPUT
	utility_error														: STRING;
    /// <summary>XV10</summary>
	dead_air_inlet_valve_clear											: BOOL;
    /// <summary>XV11</summary>
	product_line_ambient_valve_clear									: BOOL;
    /// <summary>XV03</summary>
	vacuum_pump_inlet_valve_clear										: BOOL;
END_VAR
VAR

	fbWriteData															: FB_WritePersistentData;
	tonWriteData														: TON;
	bWriteData															: BOOL;
	
	sError																: STRING;
	sMessage															: STRING;
	sUtilityError														: STRING;
	sRS																	: STRING;
	iAxStep																: INT;
	i2Step																: INT;
	i3Step																: INT;
	i8Step																: INT;
	i9Step																: INT;
	iVfd_Speed															: INT;
	bCondition1															: BOOL;
	bCondition2															: BOOL;
	bCondition3															: BOOL;
	bAdsorptionActive													: BOOL;
	bComplete															: BOOL;
	bPreCheckDone														: BOOL;
	bTimer																: BOOL;
	bPass1																: BOOL;
	bPass2																: BOOL;
	bPass3																: BOOL;
	bAdsorptionTimer													: BOOL;
	bCloseXVValves														: BOOL;
	bRunSteamBypass														: BOOL;
	bVfd_Speed_Up														: BOOL;
	bCondenserKnockoutError												: BOOL;
	bVacuumSeparatorFillError											: BOOL;
	bVacuumSeparatorDrainError											: BOOL;
	rTime																: REAL;
	rSP																	: REAL;
	rPres																: REAL;
	tonTimer															: TON;
	tonAdsorptionTimer													: TON;
	tonBoilerCheck														: TON;
	tonVacuumInterlock													: TON;
	tonCondenserKODrain													: TON;
	tonVacuumSeparatorFill												: TON;
	tonVacuumSeparatorDrain												: TON;
	rtrigVacuumSeparator												: R_TRIG;
	rtrigKODrainValve													: R_TRIG;
	
	bCondenserFlowError													: BOOL;
	bCondensateFlowError												: BOOL;
	bFlowCalibrationDiffPresError										: BOOL;
	bInletLineTempError                                  	            : BOOL;
	bProductOutletCo2Error												: BOOL;
	bProductOutletFlowError												: BOOL;
	bProductOutletH2oError												: BOOL;
	bProductTempError                                   		       	: BOOL;
	bProductVacuumPresError												: BOOL;
	bProductVacuumTempError                              	          	: BOOL;
	bSteamFlowError														: BOOL;
	bSteamLinePresError													: BOOL;
	bSteamWaterTankLevelError											: BOOL;
	bVacuumPumpWaterFlowError											: BOOL;
	bVacuumPumpWaterTemp1Error											: BOOL;
	bVacuumSeparatorLevelError											: BOOL;
	bWaterFeedFlowError													: BOOL;
	bWaterScale1Error													: BOOL;
	bWaterScale2Error													: BOOL;
	bWaterScale3Error													: BOOL;

	fb_Vacuum_Pres_Control_Valve_PI										: FB_PI_Control();
	fb_Steam_Flow_Control_Valve_PI										: FB_PI_Control();
	
	fb_WaterScales_In													: FB_RateOfChange;
 	fb_WaterScales_Out													: FB_RateOfChange;
	{attribute 'OPC.UA.DA' := '1'} 
	water_scales_in_delta												: REAL;
	{attribute 'OPC.UA.DA' := '1'} 
	water_scales_out_delta												: REAL;
	{attribute 'OPC.UA.DA' := '1'} 
	water_scales_in_rate												: REAL;
	{attribute 'OPC.UA.DA' := '1'} 
	water_scales_out_rate												: REAL;
	{attribute 'OPC.UA.DA' := '1'} 
	water_scales_reset													: BOOL;
	fb_adsorp_product_wastewater										: FB_ChangeOfValue;
	
	{attribute 'OPC.UA.DA' := '1'}  				                
	pressure_drop_test													: BOOL;							// Pressure drop test flag

	{attribute 'OPC.UA.DA' := '1'}  				                
	interlock_condenser_steam_or										: BOOL;							// Override condenser pump & fan needing to be on when steam is flowing
	{attribute 'OPC.UA.DA' := '1'}  				                
	{attribute 'OPC.UA.DA.Access' := '1'}  				                
	interlock_condenser_steam_or_status									: BOOL;
	{attribute 'OPC.UA.DA' := '1'}  				                
	{attribute 'OPC.UA.DA.Access' := '1'}  				                
	condenser_steam_interlock											: BOOL;
	
	{attribute 'OPC.UA.DA' := '1'}  				                
	interlock_hot_reactor_condenser_or									: BOOL;							// Override dead air valve needing to be open if sorbent temp is high
	{attribute 'OPC.UA.DA' := '1'}  				                
	{attribute 'OPC.UA.DA.Access' := '1'}  				                
	interlock_hot_reactor_condenser_or_status							: BOOL;
	
	{attribute 'OPC.UA.DA' := '1'}  				                
	interlock_no_steam_unevacuated_reactor_or							: BOOL;							// Override no steam to unevacuated reactor
	{attribute 'OPC.UA.DA' := '1'}  				                
	{attribute 'OPC.UA.DA.Access' := '1'}  				                
	interlock_no_steam_unevacuated_reactor_or_status					: BOOL;
	
	{attribute 'OPC.UA.DA' := '1'}  				                
	interlock_cooling_with_vacuum_or									: BOOL;							// Override vacuum not running without cooling loop active
	{attribute 'OPC.UA.DA' := '1'}  				                
	{attribute 'OPC.UA.DA.Access' := '1'}  				                
	interlock_cooling_with_vacuum_or_status								: BOOL;
	{attribute 'OPC.UA.DA' := '1'}  				                
	{attribute 'OPC.UA.DA.Access' := '1'}  				                
	cooling_with_vacuum_interlock										: BOOL;
	
	{attribute 'OPC.UA.DA' := '1'}  				                
	interlock_separator_water_level_with_vacuum_or						: BOOL;							// Override vacuum not running while separator water level too high or too low
	{attribute 'OPC.UA.DA' := '1'}  				                
	{attribute 'OPC.UA.DA.Access' := '1'}  				                
	interlock_separator_water_level_with_vacuum_or_status				: BOOL;
	{attribute 'OPC.UA.DA' := '1'}  				                
	{attribute 'OPC.UA.DA.Access' := '1'}  				                
	separator_water_level_with_vacuum_interlock							: BOOL;
	
	{attribute 'OPC.UA.DA' := '1'}  				                
	interlock_cooling_loop_flow_with_vacuum_or							: BOOL;							// Override vacuum not running with insufficient cooling flow
	{attribute 'OPC.UA.DA' := '1'}  				                
	{attribute 'OPC.UA.DA.Access' := '1'}  				                
	interlock_cooling_loop_flow_with_vacuum_or_status					: BOOL;
	{attribute 'OPC.UA.DA' := '1'}  				                
	{attribute 'OPC.UA.DA.Access' := '1'}  				                
	cooling_loop_flow_with_vacuum_interlock								: BOOL;
	
	{attribute 'OPC.UA.DA' := '1'}  				                
	interlock_condensate_tank_level_for_steam_or						: BOOL;							// Override steam not running with condensate collection tank low 
	{attribute 'OPC.UA.DA' := '1'}  				                
	{attribute 'OPC.UA.DA.Access' := '1'}  				                
	interlock_condensate_tank_level_for_steam_or_status					: BOOL;
	{attribute 'OPC.UA.DA' := '1'}  				                
	{attribute 'OPC.UA.DA.Access' := '1'}  				                
	condensate_tank_level_for_steam_interlock							: BOOL;
	
	{attribute 'OPC.UA.DA' := '1'}  				                
	interlock_hot_sorbent_for_repressurization_or						: BOOL;							// Override repressurization not running if sorbent temp is high 
	{attribute 'OPC.UA.DA' := '1'}  				                
	{attribute 'OPC.UA.DA.Access' := '1'}  				                
	interlock_hot_sorbent_for_repressurization_or_status				: BOOL;
	
	{attribute 'OPC.UA.DA' := '1'}  				                
	interlock_reactor_over_safe_pressure_limit_or						: BOOL;							// Override reactor over safe pressure limit
	{attribute 'OPC.UA.DA' := '1'}  				                
	{attribute 'OPC.UA.DA.Access' := '1'}  				                
	interlock_reactor_over_safe_pressure_limit_or_status				: BOOL;
	
	{attribute 'OPC.UA.DA' := '1'}  				                
	interlock_reactor_over_safe_temperature_limit_or					: BOOL;							// Override reactor over safe temperature limit
	{attribute 'OPC.UA.DA' := '1'}  				                
	{attribute 'OPC.UA.DA.Access' := '1'}  				                
	interlock_reactor_over_safe_temperature_limit_or_status				: BOOL;
	
	{attribute 'OPC.UA.DA' := '1'}  				                
	interlock_repressurization_valve_with_steam_or						: BOOL;							// Override repressurization valve with steam flow
	{attribute 'OPC.UA.DA' := '1'}  				                
	{attribute 'OPC.UA.DA.Access' := '1'}  				                
	interlock_repressurization_valve_with_steam_or_status				: BOOL;
	
	{attribute 'OPC.UA.DA' := '1'}  				                
	interlock_door_open_with_steam_flow_or								: BOOL;							// Override door open with steam flow
	{attribute 'OPC.UA.DA' := '1'}  				                
	{attribute 'OPC.UA.DA.Access' := '1'}  				                
	interlock_door_open_with_steam_flow_or_status						: BOOL;
	
	{attribute 'OPC.UA.DA' := '1'}  				                
	interlock_door_open_with_reactor_vacuum_or							: BOOL;							// Override door open with reactor under vacuum
	{attribute 'OPC.UA.DA' := '1'}  				                
	{attribute 'OPC.UA.DA.Access' := '1'}  				                
	interlock_door_open_with_reactor_vacuum_or_status					: BOOL;
	
	{attribute 'OPC.UA.DA' := '1'}  				                
	interlock_co2_adsorption_or											: BOOL;							// Override co2 adsorption solenoids
	{attribute 'OPC.UA.DA' := '1'}  				                
	{attribute 'OPC.UA.DA.Access' := '1'}  				                
	interlock_co2_adsorption_or_status									: BOOL;
	
	{attribute 'OPC.UA.DA' := '1'}  				                
	interlock_condensate_pump_or										: BOOL;							// Override condensate pump
	{attribute 'OPC.UA.DA' := '1'}  				                
	{attribute 'OPC.UA.DA.Access' := '1'}  				                
	interlock_condensate_pump_or_status									: BOOL;
	{attribute 'OPC.UA.DA' := '1'}  				                
	{attribute 'OPC.UA.DA.Access' := '1'}  				                
	interlock_condensate_pump											: BOOL;
	
	{attribute 'OPC.UA.DA' := '1'}  				                
	vacuum_separator_drain_or_on										: BOOL;
	{attribute 'OPC.UA.DA' := '1'}  				                
	{attribute 'OPC.UA.DA.Access' := '1'}  				                
	vacuum_separator_drain_or_on_status									: BOOL;
	{attribute 'OPC.UA.DA' := '1'}  				                
	vacuum_separator_drain_or_off										: BOOL;
	{attribute 'OPC.UA.DA' := '1'}  				                
	{attribute 'OPC.UA.DA.Access' := '1'}  				                
	vacuum_separator_drain_or_off_status								: BOOL;

	{attribute 'OPC.UA.DA' := '1'}  				                
	reactor_drain_or_on													: BOOL;
	{attribute 'OPC.UA.DA' := '1'}  				                
	{attribute 'OPC.UA.DA.Access' := '1'}  				                
	reactor_drain_or_on_status											: BOOL;
	{attribute 'OPC.UA.DA' := '1'}  				                
	reactor_drain_or_off												: BOOL;
	{attribute 'OPC.UA.DA' := '1'}  				                
	{attribute 'OPC.UA.DA.Access' := '1'}  				                
	reactor_drain_or_off_status											: BOOL;

	{attribute 'OPC.UA.DA' := '1'}  				                
	condenser_knockout_drain_or_on										: BOOL;
	{attribute 'OPC.UA.DA' := '1'}  				                
	{attribute 'OPC.UA.DA.Access' := '1'}  				                
	condenser_knockout_drain_or_on_status								: BOOL;
	{attribute 'OPC.UA.DA' := '1'}  				                
	condenser_knockout_drain_or_off										: BOOL;
	{attribute 'OPC.UA.DA' := '1'}  				                
	{attribute 'OPC.UA.DA.Access' := '1'}  				                
	condenser_knockout_drain_or_off_status								: BOOL;

	{attribute 'OPC.UA.DA' := '1'}  				                
	{attribute 'OPC.UA.DA.Access' := '1'}  				                
	warmup_complete														: BOOL;
	{attribute 'OPC.UA.DA' := '1'}  				                
	{attribute 'OPC.UA.DA.Access' := '1'}  				                
	steam_bypass_complete												: BOOL;

	{attribute 'OPC.UA.DA' := '1'}  				                
	write_persistent_data												: BOOL;
	{attribute 'OPC.UA.DA' := '1'}  				                
	drainage_function_on_or												: BOOL;
	{attribute 'OPC.UA.DA' := '1'}  				                
	drainage_function_off_or											: BOOL;
	
	
	// PIDs
	steam_valve_pid 												: FB_CTRL_PID;
	steam_valve_pid_params											: ST_CTRL_PID_PARAMS;
	steam_valve_pid_mode											: E_CTRL_MODE := E_CTRL_MODE.eCTRL_MODE_MANUAL;
	steam_valve_pid_manual_sp										: LREAL := 50;   // Pressure SP value in manual mode
	steam_valve_pid_sp_value										: LREAL;  // Pressure SP value
	steam_valve_pid_actual_value									: LREAL;  // Presure Actual Value
	steam_valve_pid_out												: LREAL;  // valve control signal ( 0-100 %)
	steam_valve_pid_simulate_timer									: TON;
	steam_valve_pid_kp												: LREAL := 0.5;
	steam_valve_pid_tn												: TIME := T#5S;
	steam_valve_pid_tv												: TIME := T#0S;
	
	
	simulate_process												: FB_CTRL_PT2oscillation;
	simulate_process_params											: ST_CTRL_PT2oscillation_PARAMS ;
	simulate_process_kp												: REAL := 20;
	simulate_process_dumping_ration									: REAL := 0.5;
	simulate_process_tT0											: REAL := 0;
	
//	fb_MovingAverage												: FB_CTRL_MOVING_AVERAGE;
	moving_avg_in													: REAL;
	moving_avg_out													: LREAL;
	moving_avg_params												: ST_CTRL_MOVING_AVERAGE_PARAMS;
	moving_avg_array												: ARRAY[1..10] OF REAL;
	moving_avg_in_sim_timer											: TON;
	
	fbMovingAverage													: FB_MovingAverage;
	
	condenser_tank_capacity										: REAL;
	steam_delivery_tank_capacity										: REAL;
	condenser_tank_room_before_full										: REAL;
	steam_delivery_tank_before_empty										: REAL;
	
    /// <summary>LS01</summary>
	{attribute 'OPC.UA.DA' := '1'}  				                
	{attribute 'OPC.UA.DA.Access' := '1'}  				                
	product_condensate_drum_lsl									AT %I*	: BOOL;
    /// <summary>LS02</summary>
	{attribute 'OPC.UA.DA' := '1'}  				                
	{attribute 'OPC.UA.DA.Access' := '1'}  				                
	product_condensate_drum_lsh									AT %I*	: BOOL;

    /// <summary>B01</summary>
	{attribute 'OPC.UA.DA' := '1'}  				                
	{attribute 'OPC.UA.DA.Access' := '1'}  				                
	boiler_package_cmd_status											: BOOL;
    /// <summary>B01</summary>
	{attribute 'OPC.UA.DA' := '1'}  				                
	boiler_ready														: BOOL;
    /// <summary>boiler package</summary>
	B_01														AT %Q*	: BOOL;
    /// <summary>B01</summary>
	{attribute 'OPC.UA.DA' := '1'}  				                
	boiler_reset												AT %Q*	: BOOL;
	
    /// <summary>P02</summary>
	{attribute 'OPC.UA.DA' := '1'}  				                
	{attribute 'OPC.UA.DA.Access' := '1'}  				                
	steam_water_pump_cmd_status											: BOOL;
    /// <summary>vacuum pump</summary>
	P_01														AT %Q*	: BOOL;

    /// <summary>P02</summary>
	{attribute 'OPC.UA.DA' := '1'}  				                
	{attribute 'OPC.UA.DA.Access' := '1'}  				                
	vacuum_pump_cmd_status												: BOOL;
    /// <summary>vacuum pump</summary>
	P_02														AT %Q*	: BOOL;

    /// <summary>P03</summary>
	{attribute 'OPC.UA.DA' := '1'}  				                
	condensate_pump														: BOOL;
    /// <summary>P03</summary>
	{attribute 'OPC.UA.DA' := '1'}  				                
	{attribute 'OPC.UA.DA.Access' := '1'}  				                
	condensate_pump_cmd_status											: BOOL;
    /// <summary>condensate pump</summary>
	P_03														AT %Q*	: BOOL;

    /// <summary>P04</summary>
	{attribute 'OPC.UA.DA' := '1'}  				                
	{attribute 'OPC.UA.DA.Access' := '1'}  				                
	condenser_pump_cmd_status											: BOOL;
    /// <summary>condenser pump</summary>
	P_04														AT %Q*	: BOOL;

    /// <summary>P05</summary>
	{attribute 'OPC.UA.DA' := '1'}  				                
	{attribute 'OPC.UA.DA.Access' := '1'}  				                
	vacuum_liquid_pump_cmd_status										: BOOL;
    /// <summary>vacuum liquid pump</summary>
	P_05														AT %Q*	: BOOL;

    /// <summary>P06</summary>
	{attribute 'OPC.UA.DA' := '1'}  				                
	{attribute 'OPC.UA.DA.Access' := '1'}  				                
	vacuum_separator_drain_pump_cmd_status								: BOOL;
    /// <summary>vacuum cooling pump</summary>
	P_06														AT %Q*	: BOOL;

    /// <summary>E01</summary>
	{attribute 'OPC.UA.DA' := '1'}  				                
	{attribute 'OPC.UA.DA.Access' := '1'}  				                
	condenser_fan_cmd_status											: BOOL;
    /// <summary>condenser fan</summary>
	E_01														AT %Q*	: BOOL;

    /// <summary>X01</summary>
	{attribute 'OPC.UA.DA' := '1'}  				                
	{attribute 'OPC.UA.DA.Access' := '1'}  				                
	vacuum_liquid_loop_fan_cmd_status									: BOOL;
    /// <summary>vacuum liquid loop fan</summary>
	X_01														AT %Q*	: BOOL;

    /// <summary>AT02</summary>
	{attribute 'OPC.UA.DA' := '1'}  				                
	{attribute 'OPC.UA.DA.Access' := '1'}  				                
	product_outlet_co2													: REAL;
	{attribute 'OPC.UA.DA' := '1'}  				                
	{attribute 'OPC.UA.DA.Access' := '1'} 
    /// <summary>AT02</summary>
	product_outlet_co2_error											: BOOL;
    /// <summary>product outlet co2</summary>
	{attribute 'OPC.UA.DA' := '1'}  				                
	_ProductOutletCO2ErrorOff											: BOOL;
    /// <summary>AT02</summary>
	{attribute 'OPC.UA.DA' := '1'}  				                
	AT_02														AT %I*	: INT;
    /// <summary>AT02</summary>
	{attribute 'OPC.UA.DA' := '1'}  				                
	{attribute 'OPC.UA.DA.Access' := '1'}  				                
	AT_02_error													AT %I*	: BOOL;
    
	/// <summary>AT03</summary>
	{attribute 'OPC.UA.DA' := '1'}  				                
	{attribute 'OPC.UA.DA.Access' := '1'}  				                
	product_outlet_h2o													: REAL;
    /// <summary>AT03</summary>
	{attribute 'OPC.UA.DA' := '1'}  				                
	{attribute 'OPC.UA.DA.Access' := '1'}  				                
	product_outlet_h2o_error											: BOOL;
	/// <summary>AT03</summary>
	{attribute 'OPC.UA.DA' := '1'}  				                
	_ProductOutletH2OErrorOff											: BOOL;
    /// <summary>product outlet h2o</summary>
	AT_03														AT %I*	: INT;
    /// <summary>product outlet h2o</summary>
	{attribute 'OPC.UA.DA' := '1'}  				                
	{attribute 'OPC.UA.DA.Access' := '1'}  				                
	AT_03_error													AT %I*	: BOOL;

    /// <summary>FT02</summary>
	{attribute 'OPC.UA.DA' := '1'}  				                
	{attribute 'OPC.UA.DA.Access' := '1'}  					                
	product_outlet_flow													: REAL;
    /// <summary>FT02</summary>
	{attribute 'OPC.UA.DA' := '1'}  				                
	{attribute 'OPC.UA.DA.Access' := '1'}  				                
	product_outlet_flow_error											: BOOL;
    /// <summary>FT02</summary>
	{attribute 'OPC.UA.DA' := '1'}  				                
	_ProductOutletFlowErrorOff											: BOOL;
    /// <summary>product outlet flow</summary>
	FT_02														AT %I*	: INT;
    /// <summary>product outlet flow</summary>
	{attribute 'OPC.UA.DA' := '1'}  				                
	{attribute 'OPC.UA.DA.Access' := '1'}  				                
	FT_02_error													AT %I*	: BOOL;

    /// <summary>FT04</summary>
	{attribute 'OPC.UA.DA' := '1'}  				                
	{attribute 'OPC.UA.DA.Access' := '1'}  				                
	condensate_flow														: REAL;
    /// <summary>FT04</summary>
	{attribute 'OPC.UA.DA' := '1'}  				                
	{attribute 'OPC.UA.DA.Access' := '1'}  				                
	condensate_flow_error												: BOOL;
    /// <summary>FT04</summary>
	{attribute 'OPC.UA.DA' := '1'}  				                
	_CondensateFlowErrorOff												: BOOL;
    /// <summary>condensate flow</summary>
	FT_04														AT %I*	: INT;
    /// <summary>condensate flow</summary>
	{attribute 'OPC.UA.DA' := '1'}  				                
	{attribute 'OPC.UA.DA.Access' := '1'}  				                
	FT_04_error													AT %I*	: BOOL;

    /// <summary>FT05</summary>
	{attribute 'OPC.UA.DA' := '1'}  				                
	{attribute 'OPC.UA.DA.Access' := '1'}  					                
	tap_water_feed_flow													: REAL;
    /// <summary>FT05</summary>
	{attribute 'OPC.UA.DA' := '1'}  				                
	{attribute 'OPC.UA.DA.Access' := '1'}  				                
	tap_water_feed_flow_error											: BOOL;
    /// <summary>FT05</summary>
	{attribute 'OPC.UA.DA' := '1'}  				                
	_TapWaterFeedFlowErrorOff											: BOOL;
    /// <summary>tap water feed flow</summary>
	FT_05														AT %I*	: INT;
    /// <summary>tap water feed flow</summary>
	{attribute 'OPC.UA.DA' := '1'}  				                
	{attribute 'OPC.UA.DA.Access' := '1'}  				                
	FT_05_error													AT %I*	: BOOL;

    /// <summary>FT06</summary>
	{attribute 'OPC.UA.DA' := '1'}  				                
	{attribute 'OPC.UA.DA.Access' := '1'}  					                
	steam_flow															: REAL;
    /// <summary>FT06</summary>
	{attribute 'OPC.UA.DA' := '1'}  				                
	{attribute 'OPC.UA.DA.Access' := '1'}  				                
	steam_flow_error													: BOOL;
    /// <summary>FT06</summary>
	{attribute 'OPC.UA.DA' := '1'}  				                
	_SteamFlowErrorOff													: BOOL;
    /// <summary>steam flow</summary>
	FT_06														AT %I*	: INT;
    /// <summary>steam flow</summary>
	{attribute 'OPC.UA.DA' := '1'}  				                
	{attribute 'OPC.UA.DA.Access' := '1'}  				                
	FT_06_error													AT %I*	: BOOL;

    /// <summary>FT07</summary>
	{attribute 'OPC.UA.DA' := '1'}  				                
	{attribute 'OPC.UA.DA.Access' := '1'}  					                
	vacuum_pump_water_flow												: REAL;
    /// <summary>FT07</summary>
	{attribute 'OPC.UA.DA' := '1'}  				                
	{attribute 'OPC.UA.DA.Access' := '1'}  				                
	vacuum_pump_water_flow_error										: BOOL;
    /// <summary>FT07</summary>
	{attribute 'OPC.UA.DA' := '1'}  				                
	_VacuumPumpWaterFlowErrorOff										: BOOL;
    /// <summary>vacuum pump water flow</summary>
	FT_07														AT %I*	: INT;
    /// <summary>vacuum pump water flow</summary>
    /// <summary>FT07</summary>
	{attribute 'OPC.UA.DA' := '1'}  				                
	{attribute 'OPC.UA.DA.Access' := '1'}  				                
	FT_07_error													AT %I*	: BOOL;

    /// <summary>FT08</summary>
	{attribute 'OPC.UA.DA' := '1'}  				                
	{attribute 'OPC.UA.DA.Access' := '1'}  					                
	condenser_flow														: REAL;
    /// <summary>FT08</summary>
	{attribute 'OPC.UA.DA' := '1'}  				                
	{attribute 'OPC.UA.DA.Access' := '1'}  				                
	condenser_flow_error												: BOOL;
    /// <summary>FT08</summary>
	{attribute 'OPC.UA.DA' := '1'}  				                
	_CondenserFlowErrorOff												: BOOL;
    /// <summary>vacuum pump water flow</summary>
	FT_08														AT %I*	: INT;
    /// <summary>vacuum pump water flow</summary>
    /// <summary>FT08</summary>
	{attribute 'OPC.UA.DA' := '1'}  				                
	{attribute 'OPC.UA.DA.Access' := '1'}  				                
	FT_08_error													AT %I*	: BOOL;

    /// <summary>LT01</summary>
	{attribute 'OPC.UA.DA' := '1'}  				                
	{attribute 'OPC.UA.DA.Access' := '1'}  					                
	steam_water_tank_level												: REAL;
    /// <summary>LT01</summary>
	{attribute 'OPC.UA.DA' := '1'}  				                
	{attribute 'OPC.UA.DA.Access' := '1'}  				                
	steam_water_tank_level_error										: BOOL;
    /// <summary>LT01</summary>
	{attribute 'OPC.UA.DA' := '1'}  				                
	_SteamWaterTankLevelErrorOff										: BOOL;
    /// <summary>steam water tank level</summary>
	LT_01														AT %I*	: INT;
    /// <summary>steam water tank level</summary>
    /// <summary>LT01</summary>
	{attribute 'OPC.UA.DA' := '1'}  				                
	{attribute 'OPC.UA.DA.Access' := '1'}  				                
	LT_01_error													AT %I*	: BOOL;

    /// <summary>LT02</summary>
	{attribute 'OPC.UA.DA' := '1'}  				                
	{attribute 'OPC.UA.DA.Access' := '1'}  					                
	vacuum_separator_level												: REAL;
    /// <summary>LT02</summary>
	{attribute 'OPC.UA.DA' := '1'}  				                
	{attribute 'OPC.UA.DA.Access' := '1'}  				                
	vacuum_separator_level_error										: BOOL;
    /// <summary>LT02</summary>
	{attribute 'OPC.UA.DA' := '1'}  				                
	_VacuumSeparatorLevelErrorOff										: BOOL;
    /// <summary>vacuum separator level</summary>
	LT_02														AT %I*	: INT;
    /// <summary>vacuum separator level</summary>
    /// <summary>LT02</summary>
	{attribute 'OPC.UA.DA' := '1'}  				                
	{attribute 'OPC.UA.DA.Access' := '1'}  				                
	LT_02_error													AT %I*	: BOOL;

    /// <summary>PT04</summary>
	{attribute 'OPC.UA.DA' := '1'}  				                
	{attribute 'OPC.UA.DA.Access' := '1'}  				                
	product_vacuum_pres													: REAL;
    /// <summary>PT04</summary>
	{attribute 'OPC.UA.DA' := '1'}  				                
	{attribute 'OPC.UA.DA.Access' := '1'}  				                
	product_vacuum_pres_error											: BOOL;
    /// <summary>PT04</summary>
	{attribute 'OPC.UA.DA' := '1'}  				                
	_ProductVacuumPresErrorOff											: BOOL;
    /// <summary>product vacuum pres</summary>
	PT_04														AT %I*	: INT;
    /// <summary>product vacuum pres</summary>
    /// <summary>PT04</summary>
	{attribute 'OPC.UA.DA' := '1'}  				                
	{attribute 'OPC.UA.DA.Access' := '1'}  				                
	PT_04_error													AT %I*	: BOOL;

    /// <summary>PT07</summary>
	{attribute 'OPC.UA.DA' := '1'}  				                
	{attribute 'OPC.UA.DA.Access' := '1'}  				                
	steam_line_pres														: REAL;
    /// <summary>PT07</summary>
	{attribute 'OPC.UA.DA' := '1'}  				                
	{attribute 'OPC.UA.DA.Access' := '1'}  				                
	steam_line_pres_error												: BOOL;
    /// <summary>PT07</summary>
	{attribute 'OPC.UA.DA' := '1'}  				                
	_SteamLinePresErrorOff												: BOOL;
    /// <summary>steam line pres</summary>
	PT_07														AT %I*	: INT;
    /// <summary>steam line pres</summary>
	{attribute 'OPC.UA.DA' := '1'}  				                
	{attribute 'OPC.UA.DA.Access' := '1'}  				                
	PT_07_error													AT %I*	: BOOL;

    /// <summary>PDT04</summary>
	{attribute 'OPC.UA.DA' := '1'}  				                
	{attribute 'OPC.UA.DA.Access' := '1'}  				                
	flow_calibration_diff_pres											: REAL;
    /// <summary>PDT04</summary>
	{attribute 'OPC.UA.DA' := '1'}  				                
	{attribute 'OPC.UA.DA.Access' := '1'}  				                
	flow_calibration_diff_pres_error									: BOOL;
    /// <summary>PDT04</summary>
	{attribute 'OPC.UA.DA' := '1'}  				                
	_FlowCalibrationDiffPresErrorOff									: BOOL;
    /// <summary>flow calibration diff pres</summary>
	PDT_04														AT %I*	: INT;
    /// <summary>flow calibration diff pres</summary>
	{attribute 'OPC.UA.DA' := '1'}  				                
	{attribute 'OPC.UA.DA.Access' := '1'}  				                
	PDT_04_error												AT %I*	: BOOL;

    /// <summary>TT02</summary>
	{attribute 'OPC.UA.DA' := '1'}  				                
	{attribute 'OPC.UA.DA.Access' := '1'}  				                
	product_temp														: REAL;
    /// <summary>TT02</summary>
	{attribute 'OPC.UA.DA' := '1'}  				                
	{attribute 'OPC.UA.DA.Access' := '1'}  				                
	product_temp_error													: BOOL;
	{attribute 'OPC.UA.DA' := '1'}  				                
	_ProductTempErrorOff												: BOOL;
    /// <summary>product temp</summary>
	TT_02														AT %I*	: INT;
    /// <summary>product temp</summary>
	{attribute 'OPC.UA.DA' := '1'}  				                
	{attribute 'OPC.UA.DA.Access' := '1'}  				                
	TT_02_error													AT %I*	: BOOL;

    /// <summary>TT03</summary>
	{attribute 'OPC.UA.DA' := '1'}  				                
	{attribute 'OPC.UA.DA.Access' := '1'}  				                
	product_vacuum_temp													: REAL;
    /// <summary>TT03</summary>
	{attribute 'OPC.UA.DA' := '1'}  				                
	{attribute 'OPC.UA.DA.Access' := '1'}  				                
	product_vacuum_temp_error											: BOOL;
    /// <summary>TT03</summary>
	{attribute 'OPC.UA.DA' := '1'}  				                
	_ProductVacuumTempOff												: BOOL;
    /// <summary>product vacuum temp</summary>
	TT_03														AT %I*	: INT;
    /// <summary>product vacuum temp</summary>
	{attribute 'OPC.UA.DA' := '1'}  				                
	{attribute 'OPC.UA.DA.Access' := '1'}  				                
	TT_03_error													AT %I*	: BOOL;

    /// <summary>TT06</summary>
	{attribute 'OPC.UA.DA' := '1'}  				                
	{attribute 'OPC.UA.DA.Access' := '1'}  				                
	inlet_line_temp														: REAL;
    /// <summary>TT06</summary>
	{attribute 'OPC.UA.DA' := '1'}  				                
	{attribute 'OPC.UA.DA.Access' := '1'}  				                
	inlet_line_temp_error												: BOOL;
    /// <summary>TT06</summary>
	{attribute 'OPC.UA.DA' := '1'}  				                
	_InletLineTempErrorOff												: BOOL;
    /// <summary>inlet line temp</summary>
	TT_06														AT %I*	: INT;
    /// <summary>inlet line temp</summary>
	{attribute 'OPC.UA.DA' := '1'}  				                
	{attribute 'OPC.UA.DA.Access' := '1'}  				                
	TT_06_error													AT %I*	: BOOL;

    /// <summary>TT10</summary>
	{attribute 'OPC.UA.DA' := '1'}  				                
	{attribute 'OPC.UA.DA.Access' := '1'}  				                
	vacuum_pump_water_temp_1											: REAL;
    /// <summary>TT10</summary>
	{attribute 'OPC.UA.DA' := '1'}  				                
	{attribute 'OPC.UA.DA.Access' := '1'}  				                
	vacuum_pump_water_temp_1_error										: BOOL;
    /// <summary>TT10</summary>
	{attribute 'OPC.UA.DA' := '1'}  				                
	_VacuumPumpWaterTemp1ErrorOff										: BOOL;
    /// <summary>vacuum pump water temp 1</summary>
	TT_10														AT %I*	: INT;
    /// <summary>vacuum pump water temp 1</summary>
	{attribute 'OPC.UA.DA' := '1'}  				                
	{attribute 'OPC.UA.DA.Access' := '1'}  				                
	TT_10_error													AT %I*	: BOOL;
	
    /// <summary>TT11</summary>
	{attribute 'OPC.UA.DA' := '1'}  				                
	{attribute 'OPC.UA.DA.Access' := '1'}  				                
	vacuum_pump_water_temp_2											: REAL;
    /// <summary>TT11</summary>
	{attribute 'OPC.UA.DA' := '1'}  				                
	{attribute 'OPC.UA.DA.Access' := '1'}  				                
	vacuum_pump_water_temp_2_error										: BOOL;
    /// <summary>TT11</summary>
	{attribute 'OPC.UA.DA' := '1'}  				                
	_VacuumPumpWaterTemp2ErrorOff										: BOOL;
    /// <summary>vacuum pump water temp 2</summary>
	TT_11														AT %I*	: INT;
    /// <summary>vacuum pump water temp 2</summary>
	{attribute 'OPC.UA.DA' := '1'}  				                
	{attribute 'OPC.UA.DA.Access' := '1'}  				                
	TT_11_error													AT %I*	: BOOL;

    /// <summary>XV03</summary>
	{attribute 'OPC.UA.DA' := '1'}  				                
	{attribute 'OPC.UA.DA.Access' := '1'}  				                
	vacuum_pump_inlet_valve_open_cmd_status								: BOOL;
    /// <summary>XV03</summary>
	{attribute 'OPC.UA.DA' := '1'}  				                
	{attribute 'OPC.UA.DA.Access' := '1'}  				                
	vacuum_pump_inlet_valve_open								AT %I*	: BOOL;
    /// <summary>XV03</summary>
	{attribute 'OPC.UA.DA' := '1'}  				                
	{attribute 'OPC.UA.DA.Access' := '1'}  				                
	vacuum_pump_inlet_valve_closed								AT %I*	: BOOL;
    /// <summary>vacuum pump inlet valve</summary>
	XV_03														AT %Q*	: BOOL;
	
    /// <summary>XV04</summary>
	{attribute 'OPC.UA.DA' := '1'}  				                
	{attribute 'OPC.UA.DA.Access' := '1'}  				                
	vacuum_pump_bypass_valve_open_cmd_status							: BOOL;
    /// <summary>XV04</summary>
	{attribute 'OPC.UA.DA' := '1'}  				                
	{attribute 'OPC.UA.DA.Access' := '1'}  				                
	vacuum_pump_bypass_valve_open								AT %I*	: BOOL;
    /// <summary>XV04</summary>
	{attribute 'OPC.UA.DA' := '1'}  				                
	{attribute 'OPC.UA.DA.Access' := '1'}  				                
	vacuum_pump_bypass_valve_closed								AT %I*	: BOOL;
    /// <summary>vacuum pump bypass valve</summary>
	XV_04														AT %Q*	: BOOL;
    /// <summary>XV04</summary>
	vacuum_pump_bypass_valve_clear										: BOOL;
	
    /// <summary>XV06</summary>
	{attribute 'OPC.UA.DA' := '1'}  				                
	knockout_drain_valve												: BOOL;
    /// <summary>XV06</summary>
	{attribute 'OPC.UA.DA' := '1'}  				                
	{attribute 'OPC.UA.DA.Access' := '1'}  				                
	knockout_drain_valve_open_cmd_status								: BOOL;
    /// <summary>XV06</summary>
	{attribute 'OPC.UA.DA' := '1'}  				                
	{attribute 'OPC.UA.DA.Access' := '1'}  				                
	knockout_drain_valve_open									AT %I*	: BOOL;
    /// <summary>XV06</summary>
	{attribute 'OPC.UA.DA' := '1'}  				                
	{attribute 'OPC.UA.DA.Access' := '1'}  				                
	knockout_drain_valve_closed									AT %I*	: BOOL;
    /// <summary>knockout drain valve</summary>
	XV_06														AT %Q*	: BOOL;
    /// <summary>XV06</summary>
	knockout_drain_valve_clear											: BOOL;
	
    /// <summary>XV10</summary>
	{attribute 'OPC.UA.DA' := '1'}  				                
	{attribute 'OPC.UA.DA.Access' := '1'}  				                
	dead_air_inlet_valve_open_cmd_status								: BOOL;
    /// <summary>XV10</summary>
	{attribute 'OPC.UA.DA' := '1'}  				                
	{attribute 'OPC.UA.DA.Access' := '1'}  				                
	dead_air_inlet_valve_open									AT %I*	: BOOL;
    /// <summary>XV10</summary>
	{attribute 'OPC.UA.DA' := '1'}  				                
	{attribute 'OPC.UA.DA.Access' := '1'}  				                
	dead_air_inlet_valve_closed 								AT %I*	: BOOL;
    /// <summary>dead air inlet valve</summary>
	XV_10														AT %Q*	: BOOL;

    /// <summary>XV11</summary>
	{attribute 'OPC.UA.DA' := '1'}  				                
	{attribute 'OPC.UA.DA.Access' := '1'}  				                
	product_line_ambient_valve_cmd_status								: BOOL;
    /// <summary>XV11</summary>
	{attribute 'OPC.UA.DA' := '1'}  				                
	{attribute 'OPC.UA.DA.Access' := '1'}  				                
	product_line_ambient_valve_product 							AT %I*	: BOOL;				///@@@ Assuming open valve is Product
    /// <summary>XV11</summary>
	{attribute 'OPC.UA.DA' := '1'}  				                
	{attribute 'OPC.UA.DA.Access' := '1'}  				                
	product_line_ambient_valve_ambient							AT %I*	: BOOL;				///@@@ Assuming closed valve is Ambient
    /// <summary>product line ambient valve</summary>
	XV_11														AT %Q*	: BOOL;

	/// <summary>XV12</summary>
	{attribute 'OPC.UA.DA' := '1'}  				                
	tap_water_feed_valve												: BOOL;
    /// <summary>XV11</summary>
	{attribute 'OPC.UA.DA' := '1'}  				                
	{attribute 'OPC.UA.DA.Access' := '1'}  				                
	tap_water_feed_valve_cmd_status										: BOOL;
	XV_12														AT %Q*	: BOOL;

	/// <summary>XV13</summary>
	{attribute 'OPC.UA.DA' := '1'}  				                
	separator_drain_valve												: BOOL;
    /// <summary>XV13</summary>
	{attribute 'OPC.UA.DA' := '1'}  				                
	{attribute 'OPC.UA.DA.Access' := '1'}  				                
	separator_drain_valve_open_cmd_status								: BOOL;
    /// <summary>XV13</summary>
	{attribute 'OPC.UA.DA' := '1'}  				                
	{attribute 'OPC.UA.DA.Access' := '1'}  				                
	separator_drain_valve_open									AT %I*	: BOOL;
    /// <summary>XV13</summary>
	{attribute 'OPC.UA.DA' := '1'}  				                
	{attribute 'OPC.UA.DA.Access' := '1'}  				                
	separator_drain_valve_closed 								AT %I*	: BOOL;
    /// <summary>dead air inlet valve</summary>
	XV_13														AT %Q*	: BOOL;
    /// <summary>XV13</summary>
	separator_drain_valve_clear											: BOOL;

	/// <summary>XV14</summary>
	{attribute 'OPC.UA.DA' := '1'}  				                
	steam_water_reservoir_valve											: BOOL;
    /// <summary>XV14</summary>
	{attribute 'OPC.UA.DA' := '1'}  				                
	{attribute 'OPC.UA.DA.Access' := '1'}  				                
	steam_water_reservoir_valve_cmd_status								: BOOL;
    /// <summary>steam water reservoir valve</summary>
	XV_14														AT %Q*	: BOOL;

    /// <summary>PCV01</summary>
	vacuum_pres_control_valve_open										: BOOL;
    /// <summary>PCV01</summary>
	vacuum_pres_control_valve_closed									: BOOL;
    /// <summary>PCV01</summary>
	{attribute 'OPC.UA.DA' := '1'}  				                
	{attribute 'OPC.UA.DA.Access' := '1'}  				                
	vacuum_pres_control_valve_position									: REAL;
    /// <summary>PCV01</summary>
	{attribute 'OPC.UA.DA' := '1'}  				                
	{attribute 'OPC.UA.DA.Access' := '1'}  				                
	vacuum_pres_control_valve_position_error					AT %I*	: BOOL;
    /// <summary>vacuum pressure control valve</summary>
	PCV_01														AT %Q*	: INT;
    /// <summary>vacuum pressure control valve</summary>
	{attribute 'OPC.UA.DA' := '1'}  				                
	{attribute 'OPC.UA.DA.Access' := '1'}  				                
	PCV_01_position												AT %I*	: INT;
    /// <summary>PCV01</summary>                  	           
	{attribute 'OPC.UA.DA' := '1'}  				                
	{attribute 'OPC.UA.DA.Access' := '1'}  				                
	vacuum_pres_control_valve_current_mode								: INT;			
    /// <summary>PCV01</summary>                  	           
	vacuum_pres_control_valve_kp										: REAL		:= 0.01; 
    /// <summary>PCV01</summary>                  	           
	vacuum_pres_control_valve_ki										: REAL		:= 0.01;
    /// <summary>PCV01</summary>                  	           
	vacuum_pres_control_valve_loop_time									: REAL		:= 2000;
    /// <summary>PCV01</summary>                  	           
	vacuum_pres_control_valve_iband										: REAL		:= 6;
    /// <summary>PCV01</summary>                  	           
	vacuum_pres_control_valve_base										: INT		:= 13110;
    /// <summary>PCV01</summary>                  	           
	vacuum_pres_control_valve_base_adjust								: INT		:= 10;
	
    /// <summary>PCV02</summary>
	steam_flow_control_valve_open										: BOOL;
    /// <summary>PCV02</summary>
	steam_flow_control_valve_closed										: BOOL;
    /// <summary>PCV02</summary>
	{attribute 'OPC.UA.DA' := '1'}  				                
	{attribute 'OPC.UA.DA.Access' := '1'}  				                
	steam_flow_control_valve_position									: REAL;
    /// <summary>PCV02</summary>
	{attribute 'OPC.UA.DA' := '1'}  				                
	{attribute 'OPC.UA.DA.Access' := '1'}  				                
	steam_flow_control_valve_position_error								: BOOL;
    /// <summary>steam flow control valve</summary>
	PCV_02														AT %Q*	: INT;
    /// <summary>steam flow control valve</summary>
	{attribute 'OPC.UA.DA' := '1'}  				                
	{attribute 'OPC.UA.DA.Access' := '1'}  				                
	PCV_02_position												AT %I*	: INT;
    /// <summary>PCV02</summary>                  	           
	{attribute 'OPC.UA.DA' := '1'}  				                
	{attribute 'OPC.UA.DA.Access' := '1'}  				                
	steam_flow_control_valve_current_mode								: INT;			
    /// <summary>PCV02</summary>                  	           
	steam_flow_control_valve_kp											: REAL		:= 0.01; 
    /// <summary>PCV02</summary>                  	           
	steam_flow_control_valve_ki											: REAL		:= 0.01;
    /// <summary>PCV02</summary>                  	           
	steam_flow_control_valve_loop_time									: REAL		:= 2000;
    /// <summary>PCV02</summary>                  	           
	steam_flow_control_valve_iband										: REAL		:= 6;
    /// <summary>PCV02</summary>                  	           
	steam_flow_control_valve_base										: INT		:= 13110;
    /// <summary>PCV02</summary>                  	           
	steam_flow_control_valve_base_adjust								: INT		:= 10;
	
	{attribute 'OPC.UA.DA' := '1'}  				                
	{attribute 'OPC.UA.DA.Access' := '1'}  				                
	l1_current_240														: REAL;
	{attribute 'OPC.UA.DA' := '1'}  				                
	{attribute 'OPC.UA.DA.Access' := '1'}  				                
	l1_current_240_error										AT %I*	: BOOL;
	IT1															AT %I*	: INT;
	{attribute 'OPC.UA.DA' := '1'}  				                
	{attribute 'OPC.UA.DA.Access' := '1'}  				                
	l2_current_240														: REAL;
	{attribute 'OPC.UA.DA' := '1'}  				                
	{attribute 'OPC.UA.DA.Access' := '1'}  				                
	l2_current_240_error										AT %I*	: BOOL;
	IT2															AT %I*	: INT;
	{attribute 'OPC.UA.DA' := '1'}  				                
	{attribute 'OPC.UA.DA.Access' := '1'}  				                
	l3_current_240														: REAL;
	{attribute 'OPC.UA.DA' := '1'}  				                
	{attribute 'OPC.UA.DA.Access' := '1'}  				                
	l3_current_240_error										AT %I*	: BOOL;
	IT3															AT %I*	: INT;
	
	{attribute 'OPC.UA.DA' := '1'}  				                
	{attribute 'OPC.UA.DA.Access' := '1'}  				                
	l1_voltage_240														: REAL;
	{attribute 'OPC.UA.DA' := '1'}  				                
	{attribute 'OPC.UA.DA.Access' := '1'}  				                
	l1_voltage_240_error										AT %I*	: BOOL;
	{attribute 'OPC.UA.DA' := '1'}  				                
	VT1															AT %I*	: INT;
	{attribute 'OPC.UA.DA' := '1'}  				                
	l2_voltage_240														: REAL;
	{attribute 'OPC.UA.DA' := '1'}  				                
	{attribute 'OPC.UA.DA.Access' := '1'}  				                
	l2_voltage_240_error										AT %I*	: BOOL;
	{attribute 'OPC.UA.DA' := '1'}  				                
	VT2															AT %I*	: INT;
	{attribute 'OPC.UA.DA' := '1'}  				                
	l3_voltage_240														: REAL;
	{attribute 'OPC.UA.DA' := '1'}  				                
	{attribute 'OPC.UA.DA.Access' := '1'}  				                
	l3_voltage_240_error										AT %I*	: BOOL;
	{attribute 'OPC.UA.DA' := '1'}  				                
	VT3															AT %I*	: INT;
	
	{attribute 'OPC.UA.DA' := '1'}  				                
	{attribute 'OPC.UA.DA.Access' := '1'}  				                
	l1_current_120														: REAL;
	{attribute 'OPC.UA.DA' := '1'}  				                
	{attribute 'OPC.UA.DA.Access' := '1'}  				                
	l1_current_120_error										AT %I*	: BOOL;
	IT4															AT %I*	: INT;
	
	{attribute 'OPC.UA.DA' := '1'}  				                
	{attribute 'OPC.UA.DA.Access' := '1'}  				                
	l1_voltage_120														: REAL;
	{attribute 'OPC.UA.DA' := '1'}  				                
	{attribute 'OPC.UA.DA.Access' := '1'}  				                
	l1_voltage_120_error										AT %I*	: BOOL;
	VT4															AT %I*	: INT;
	
	{attribute 'OPC.UA.DA' := '1'}  				                
	{attribute 'OPC.UA.DA.Access' := '1'}  				                
	l1_current_boiler													: REAL;
	{attribute 'OPC.UA.DA' := '1'}  				                
	{attribute 'OPC.UA.DA.Access' := '1'}  				                
	l1_current_boiler_error										AT %I*	: BOOL;
	IT_boiler_01												AT %I*	: INT;
	{attribute 'OPC.UA.DA' := '1'}  				                
	{attribute 'OPC.UA.DA.Access' := '1'}  				                
	l2_current_boiler													: REAL;
	{attribute 'OPC.UA.DA' := '1'}  				                
	{attribute 'OPC.UA.DA.Access' := '1'}  				                
	l2_current_boiler_error										AT %I*	: BOOL;
	IT_boiler_02												AT %I*	: INT;
	{attribute 'OPC.UA.DA' := '1'}  				                
	{attribute 'OPC.UA.DA.Access' := '1'}  				                
	l3_current_boiler													: REAL;
	{attribute 'OPC.UA.DA' := '1'}  				                
	{attribute 'OPC.UA.DA.Access' := '1'}  				                
	l3_current_boiler_error										AT %I*	: BOOL;
	IT_boiler_03												AT %I*	: INT;
	
	//== Water Scales ====
	  /// <summary>WI01</summary>
	{attribute 'OPC.UA.DA' := '1'}  				                
	{attribute 'OPC.UA.DA.Access' := '1'}  				                
	water_scale_1														: REAL;
    /// <summary>WI01</summary>
	{attribute 'OPC.UA.DA' := '1'}  				                
	{attribute 'OPC.UA.DA.Access' := '1'}  				                
	water_scale_1_error													: BOOL;
    /// <summary>WI01</summary>
	{attribute 'OPC.UA.DA' := '1'}  				                
	_WaterScale1ErrorOff												: BOOL;
    /// <summary>water scale 1</summary>
	WI_01														AT %I*	: INT;
    /// <summary>water scale 1</summary>
	{attribute 'OPC.UA.DA' := '1'}  				                
	{attribute 'OPC.UA.DA.Access' := '1'}  				                
	WI_01_error													AT %I*	: BOOL;
	
	  /// <summary>WI02</summary>
	{attribute 'OPC.UA.DA' := '1'}  				                
	{attribute 'OPC.UA.DA.Access' := '1'}  				                
	water_scale_2														: REAL;
    /// <summary>WI02</summary>
	{attribute 'OPC.UA.DA' := '1'}  				                
	{attribute 'OPC.UA.DA.Access' := '1'}  				                
	water_scale_2_error													: BOOL;
    /// <summary>WI02</summary>
	{attribute 'OPC.UA.DA' := '1'}  				                
	_WaterScale2ErrorOff												: BOOL;
    /// <summary>water scale 2</summary>
	WI_02														AT %I*	: INT;
    /// <summary>water scale 2</summary>
	{attribute 'OPC.UA.DA' := '1'}  				                
	{attribute 'OPC.UA.DA.Access' := '1'}  				                
	WI_02_error													AT %I*	: BOOL;
	
	
		  /// <summary>WI03</summary>
	{attribute 'OPC.UA.DA' := '1'}  				                
	{attribute 'OPC.UA.DA.Access' := '1'}  				                
	water_scale_3														: REAL;
    /// <summary>WI03</summary>
	{attribute 'OPC.UA.DA' := '1'}  				                
	{attribute 'OPC.UA.DA.Access' := '1'}  				                
	water_scale_3_error													: BOOL;
    /// <summary>WI03</summary>
	{attribute 'OPC.UA.DA' := '1'}  				                
	_WaterScale3ErrorOff												: BOOL;
    /// <summary>water scale 3/summary>
	WI_03														AT %I*	: INT;
    /// <summary>water scale 3</summary>
	{attribute 'OPC.UA.DA' := '1'}  				                
	{attribute 'OPC.UA.DA.Access' := '1'}  				                
	WI_03_error													AT %I*	: BOOL;
	
END_VAR

VAR PERSISTENT
	
	/// SCALING
	
    /// <summary>AT02</summary>
	{attribute 'OPC.UA.DA' := '1'}  				                
	product_outlet_co2_low												: REAL;
    /// <summary>AT02</summary>
	{attribute 'OPC.UA.DA' := '1'}  				                
	product_outlet_co2_high												: REAL;
    /// <summary>AT02</summary>
	{attribute 'OPC.UA.DA' := '1'}  				                
	product_outlet_co2_min												: REAL;
    /// <summary>AT02</summary>
	{attribute 'OPC.UA.DA' := '1'}  				                
	product_outlet_co2_offset											: REAL;
	
    /// <summary>AT03</summary>
	{attribute 'OPC.UA.DA' := '1'}  				                
	product_outlet_h2o_low												: REAL;
    /// <summary>AT03</summary>
	{attribute 'OPC.UA.DA' := '1'}  				                
	product_outlet_h2o_high												: REAL;
    /// <summary>AT03</summary>
	{attribute 'OPC.UA.DA' := '1'}  				                
	product_outlet_h2o_min												: REAL;
    /// <summary>AT03</summary>
	{attribute 'OPC.UA.DA' := '1'}  				                
	product_outlet_h2o_offset											: REAL;
	
    /// <summary>FT02</summary>
	{attribute 'OPC.UA.DA' := '1'}  				                
	product_outlet_flow_low												: REAL;
    /// <summary>FT02</summary>
	{attribute 'OPC.UA.DA' := '1'}  				                
	product_outlet_flow_high											: REAL;
    /// <summary>FT02</summary>
	{attribute 'OPC.UA.DA' := '1'}  				                
	product_outlet_flow_min												: REAL;
    /// <summary>FT02</summary>
	{attribute 'OPC.UA.DA' := '1'}  				                
	product_outlet_flow_offset											: REAL;
	
    /// <summary>FT04</summary>
	{attribute 'OPC.UA.DA' := '1'}  				                
	condensate_flow_low													: REAL;
    /// <summary>FT04</summary>
	{attribute 'OPC.UA.DA' := '1'}  				                
	condensate_flow_high												: REAL;
    /// <summary>FT04</summary>
	{attribute 'OPC.UA.DA' := '1'}  				                
	condensate_flow_min													: REAL;
    /// <summary>FT04</summary>
	{attribute 'OPC.UA.DA' := '1'}  				                
	condensate_flow_offset												: REAL;
	
    /// <summary>FT05</summary>
	{attribute 'OPC.UA.DA' := '1'}  				                
	tap_water_feed_flow_low												: REAL;
    /// <summary>FT05</summary>
	{attribute 'OPC.UA.DA' := '1'}  				                
	tap_water_feed_flow_high											: REAL;
    /// <summary>FT05</summary>
	{attribute 'OPC.UA.DA' := '1'}  				                
	tap_water_feed_flow_min												: REAL;
    /// <summary>FT05</summary>
	{attribute 'OPC.UA.DA' := '1'}  				                
	tap_water_feed_flow_offset											: REAL;

    /// <summary>FT06</summary>
	{attribute 'OPC.UA.DA' := '1'}  				                
	steam_flow_low														: REAL;
    /// <summary>FT06</summary>
	{attribute 'OPC.UA.DA' := '1'}  				                
	steam_flow_high														: REAL;
    /// <summary>FT06</summary>
	{attribute 'OPC.UA.DA' := '1'}  				                
	steam_flow_min														: REAL;
    /// <summary>FT06</summary>
	{attribute 'OPC.UA.DA' := '1'}  				                
	steam_flow_offset													: REAL;

    /// <summary>FT07</summary>
	{attribute 'OPC.UA.DA' := '1'}  				                
	vacuum_pump_water_flow_low											: REAL;
    /// <summary>FT07</summary>
	{attribute 'OPC.UA.DA' := '1'}  				                
	vacuum_pump_water_flow_high											: REAL;
    /// <summary>FT07</summary>
	{attribute 'OPC.UA.DA' := '1'}  				                
	vacuum_pump_water_flow_min											: REAL;
    /// <summary>FT07</summary>
	{attribute 'OPC.UA.DA' := '1'}  				                
	vacuum_pump_water_flow_offset										: REAL;
	
    /// <summary>FT08</summary>
	{attribute 'OPC.UA.DA' := '1'}  				                
	condenser_flow_low													: REAL;
    /// <summary>FT08</summary>
	{attribute 'OPC.UA.DA' := '1'}  				                
	condenser_flow_high													: REAL;
    /// <summary>FT08</summary>
	{attribute 'OPC.UA.DA' := '1'}  				                
	condenser_flow_min													: REAL;
    /// <summary>FT08</summary>
	{attribute 'OPC.UA.DA' := '1'}  				                
	condenser_flow_offset												: REAL;
	
    /// <summary>AT-08</summary>                        
	{attribute 'OPC.UA.DA' := '1'}  				            
	weather_wind_speed_low												: REAL;
    /// <summary>AT-08</summary>                        
	{attribute 'OPC.UA.DA' := '1'}  				            
	weather_wind_speed_high												: REAL;
    /// <summary>AT-08</summary>                        
	{attribute 'OPC.UA.DA' := '1'}  				            
	weather_wind_speed_min												: REAL;
    /// <summary>AT-08</summary>                        
	{attribute 'OPC.UA.DA' := '1'}  				            
	weather_wind_speed_offset											: REAL;
	
    /// <summary>LT01</summary>
	{attribute 'OPC.UA.DA' := '1'}  				                
	steam_water_tank_level_low											: REAL;
    /// <summary>LT01</summary>
	{attribute 'OPC.UA.DA' := '1'}  				                
	steam_water_tank_level_high											: REAL;
    /// <summary>LT01</summary>
	{attribute 'OPC.UA.DA' := '1'}  				                
	steam_water_tank_level_min											: REAL;
    /// <summary>LT01</summary>
	{attribute 'OPC.UA.DA' := '1'}  				                
	steam_water_tank_level_offset										: REAL;
	
    /// <summary>LT02</summary>
	{attribute 'OPC.UA.DA' := '1'}  				                
	vacuum_separator_level_low											: REAL;
    /// <summary>LT02</summary>
	{attribute 'OPC.UA.DA' := '1'}  				                
	vacuum_separator_level_high											: REAL;
    /// <summary>LT02</summary>
	{attribute 'OPC.UA.DA' := '1'}  				                
	vacuum_separator_level_min											: REAL;
    /// <summary>LT02</summary>
	{attribute 'OPC.UA.DA' := '1'}  				                
	vacuum_separator_level_offset										: REAL;
	
    /// <summary>PT04</summary>
	{attribute 'OPC.UA.DA' := '1'}  				                
	product_vacuum_pres_low												: REAL;
    /// <summary>PT04</summary>
	{attribute 'OPC.UA.DA' := '1'}  				                
	product_vacuum_pres_high											: REAL;
    /// <summary>PT04</summary>
	{attribute 'OPC.UA.DA' := '1'}  				                
	product_vacuum_pres_min												: REAL;
    /// <summary>PT04</summary>
	{attribute 'OPC.UA.DA' := '1'}  				                
	product_vacuum_pres_offset											: REAL;
	
    /// <summary>PT07</summary>
	{attribute 'OPC.UA.DA' := '1'}  				                
	steam_line_pres_low													: REAL;
    /// <summary>PT07</summary>
	{attribute 'OPC.UA.DA' := '1'}  				                
	steam_line_pres_high												: REAL;
    /// <summary>PT07</summary>
	{attribute 'OPC.UA.DA' := '1'}  				                
	steam_line_pres_min													: REAL;
    /// <summary>PT07</summary>
	{attribute 'OPC.UA.DA' := '1'}  				                
	steam_line_pres_offset												: REAL;
	
    /// <summary>PDT04</summary>
	{attribute 'OPC.UA.DA' := '1'}  				                
	flow_calibration_diff_pres_low										: REAL;
    /// <summary>PDT04</summary>
	{attribute 'OPC.UA.DA' := '1'}  				                
	flow_calibration_diff_pres_high										: REAL;
    /// <summary>PDT04</summary>
	{attribute 'OPC.UA.DA' := '1'}  				                
	flow_calibration_diff_pres_min										: REAL;
    /// <summary>PDT04</summary>
	{attribute 'OPC.UA.DA' := '1'}  				                
	flow_calibration_diff_pres_offset									: REAL;
	
    /// <summary>TT-02</summary>
	{attribute 'OPC.UA.DA' := '1'}  				                
	product_temp_offset													: REAL;
	
    /// <summary>TT-03</summary>
	{attribute 'OPC.UA.DA' := '1'}  				                
	product_vacuum_temp_offset											: REAL;
	
    /// <summary>TT06</summary>
	{attribute 'OPC.UA.DA' := '1'}  				                
	inlet_line_temp_offset												: REAL;
	
    /// <summary>TT10</summary>
	{attribute 'OPC.UA.DA' := '1'}  				                
	vacuum_pump_water_temp_1_offset										: REAL;

    /// <summary>TT11</summary>
	{attribute 'OPC.UA.DA' := '1'}  				                
	vacuum_pump_water_temp_2_offset										: REAL;
	
	
	/// <summary>WI01</summary>
	{attribute 'OPC.UA.DA' := '1'}  				                
	water_scale_1_low													: REAL;
    /// <summary>WI01</summary>
	{attribute 'OPC.UA.DA' := '1'}  				                
	water_scale_1_high													: REAL;
    /// <summary>WI01</summary>
	{attribute 'OPC.UA.DA' := '1'}  				                
	water_scale_1_min													: REAL;
    /// <summary>WI01</summary>
	{attribute 'OPC.UA.DA' := '1'}  				                
	water_scale_1_offset												: REAL;
	
	
	/// <summary>WI02</summary>
	{attribute 'OPC.UA.DA' := '1'}  				                
	water_scale_2_low													: REAL;
    /// <summary>WI02</summary>
	{attribute 'OPC.UA.DA' := '1'}  				                
	water_scale_2_high													: REAL;
    /// <summary>WI02</summary>
	{attribute 'OPC.UA.DA' := '1'}  				                
	water_scale_2_min													: REAL;
    /// <summary>WI02</summary>
	{attribute 'OPC.UA.DA' := '1'}  				                
	water_scale_2_offset												: REAL;
	
	/// <summary>WI03</summary>
	{attribute 'OPC.UA.DA' := '1'}  				                
	water_scale_3_low													: REAL;
    /// <summary>WI03</summary>
	{attribute 'OPC.UA.DA' := '1'}  				                
	water_scale_3_high													: REAL;
    /// <summary>WI03</summary>
	{attribute 'OPC.UA.DA' := '1'}  				                
	water_scale_3_min													: REAL;
    /// <summary>WI02</summary>
	{attribute 'OPC.UA.DA' := '1'}  				                
	water_scale_3_offset												: REAL;
	
	/// SET POINTS
	
